// TIA Portal V18 program export: 1 tag tables, 9 data types, 14 data blocks, 112 code blocks (in call order from the OBs), 66 instance data blocks

VAR_GLOBAL   // PLC tag table "Default tag table"
   "mz encoder a" AT %I0.0 : Bool;
   "mz encoder b" AT %I0.1 : Bool;
   "my encoder a" AT %I0.2 : Bool;
   "my encoder b" AT %I0.3 : Bool;
   "mx encoder a" AT %I0.4 : Bool;
   "mx encoder b" AT %I0.5 : Bool;
   "mz up indNOK" AT %I0.6 : Bool;
   "mz down indNOK" AT %I0.7 : Bool;
   "my fwd indNOK" AT %I1.0 : Bool;
   "my rev indNOK" AT %I1.1 : Bool;
   "mx right indNOK" AT %I1.2 : Bool;
   "mx left indNOK" AT %I1.3 : Bool;
   "mo1 tilt fwd indNOK" AT %I1.4 : Bool;
   "mo1 tilt rev indNOK" AT %I1.5 : Bool;
   "na(3)" AT %I1.6 : Bool;
   "na(4)" AT %I1.7 : Bool;
   ai_reserve AT %IW100 : Int;
   "ai_reserve(1)" AT %IW102 : Int;
   hscрезерв AT %ID812 : DInt;
   "hscрезерв(1)" AT %ID816 : DInt;
   "hscрезерв(2)" AT %ID820 : DInt;
   "mz hsc" AT %ID800 : DInt;
   "my hsc" AT %ID804 : DInt;
   "mx hsc" AT %ID808 : DInt;
   "a1_com_di50.0" AT %I50.0 : Bool;
   "a1_com_di50.1" AT %I50.1 : Bool;
   "a1_com_di50.2" AT %I50.2 : Bool;
   "a1_com_di50.3" AT %I50.3 : Bool;
   "a1_com_di50.4" AT %I50.4 : Bool;
   "a1_com_di50.5" AT %I50.5 : Bool;
   "a1_com_di50.6" AT %I50.6 : Bool;
   "a1_com_di50.7" AT %I50.7 : Bool;
   a1_com_di_byte AT %IB50 : Byte;
   "mo1 enc a" AT %I2.0 : Bool;
   "mo1 enc b" AT %I2.1 : Bool;
   "mo2 enc a" AT %I2.2 : Bool;
   "mo2 enc b" AT %I2.3 : Bool;
   "door enc a" AT %I2.4 : Bool;
   "door enc b" AT %I2.5 : Bool;
   "door closed 1 ind NOT" AT %I2.6 : Bool;
   "door open NOK 1 ind" AT %I2.7 : Bool;
   "res i" AT %I3.0 : Bool;
   "mo2 rot home ind" AT %I3.1 : Bool;
   "res i(1)" AT %I3.2 : Bool;
   "air pres ok" AT %I3.3 : Bool;
   "door closed 1 mech Excluded For Xray" AT %I3.4 : Bool;
   "door open 1 mech" AT %I3.5 : Bool;
   "na(1)" AT %I3.6 : Bool;
   "na(2)" AT %I3.7 : Bool;
   "ai_reserve(2)" AT %IW110 : Int;
   "ai_reserve(3)" AT %IW112 : Int;
   "hscрезерв(3)" AT %ID862 : DInt;
   "hscрезерв(4)" AT %ID866 : DInt;
   "hscрезерв(5)" AT %ID870 : DInt;
   "mo1 hsc" AT %ID850 : DInt;
   "mo2 hsc" AT %ID854 : DInt;
   "door hsc" AT %ID858 : DInt;
   "mz up mech" AT %I4.0 : Bool;
   "mz down mech" AT %I4.1 : Bool;
   "CAB phase check OK" AT %I4.2 : Bool;
   lightBarrierOK AT %I4.3 : Bool;
   "my fwd mech" AT %I4.4 : Bool;
   "my rev mech" AT %I4.5 : Bool;
   "xray coler ok" AT %I4.6 : Bool;
   ESTOP_AND_KEY_OK AT %I4.7 : Bool;
   "mx right mech" AT %I5.0 : Bool;
   "mx left mech" AT %I5.1 : Bool;
   "door closed 2 mech Excluded For Xray" AT %I5.2 : Bool;
   "door open 2 mech" AT %I5.3 : Bool;
   "mo1 tilt fwd mech" AT %I5.4 : Bool;
   "mo1 tilt rev mech" AT %I5.5 : Bool;
   "door closed 2 ind NOT" AT %I5.6 : Bool;
   "door open 2 ind NOT" AT %I5.7 : Bool;
   "desk door b close" AT %I6.0 : Bool;
   "desk door b open" AT %I6.1 : Bool;
   "desk o1 tilt b cw" AT %I6.2 : Bool;
   "desk o1 tilt b ccw" AT %I6.3 : Bool;
   "desk b home" AT %I6.4 : Bool;
   "desk b load unload" AT %I6.5 : Bool;
   "desk b laser centr" AT %I6.6 : Bool;
   "res i(3)" AT %I7.0 : Bool;
   "res i(4)" AT %I7.1 : Bool;
   ESTOP_OK AT %I7.2 : Bool;
   Y2_home_esw AT %I7.3 : Bool;
   "shutter open ind" AT %I7.5 : Bool;
   "shutter closed ind" AT %I7.4 : Bool;
   "ESTOP xray OK" AT %I7.6 : Bool;
   "res i(8)" AT %I7.7 : Bool;
   "detector safety ok" AT %I8.0 : Bool;
   "desk o2 rot b fwd" AT %I8.1 : Bool;
   "desk o2 rot b reverse" AT %I8.3 : Bool;
   "desk o2 rot b home" AT %I8.2 : Bool;
   "desk y  b rev" AT %I8.4 : Bool;
   "desk y b fwd" AT %I8.5 : Bool;
   "desk b defect next" AT %I8.6 : Bool;
   "desk b defect prev" AT %I8.7 : Bool;
   "desk sw manual" AT %I9.0 : Bool;
   "desk sw auto" AT %I9.1 : Bool;
   "desk b auto start" AT %I9.2 : Bool;
   "desk b defect mark" AT %I9.3 : Bool;
   "desk x b left" AT %I9.4 : Bool;
   "desk x b right" AT %I9.5 : Bool;
   "desk z up" AT %I9.7 : Bool;
   "desk z down" AT %I9.6 : Bool;
   "remote key activated" AT %I6.7 : Bool;
   "mz up" AT %Q0.1 : Bool;
   "mz down" AT %Q0.2 : Bool;
   "mz up STOP" AT %Q0.3 : Bool;
   "mz down STOP" AT %Q0.4 : Bool;
   "my fwd" AT %Q0.6 : Bool;
   "my rev" AT %Q0.5 : Bool;
   "my fwd STOP" AT %Q0.7 : Bool;
   "my rev STOP" AT %Q1.0 : Bool;
   "shutter out1.1" AT %Q1.1 : Bool;
   "na(5)" AT %Q1.2 : Bool;
   "na(6)" AT %Q1.3 : Bool;
   "na(7)" AT %Q1.4 : Bool;
   "na(8)" AT %Q1.5 : Bool;
   "na(9)" AT %Q1.6 : Bool;
   "na(10)" AT %Q1.7 : Bool;
   "mz up down speed" AT %QW100 : Int;
   "my fwd rev speed" AT %QW102 : Int;
   "a1_com_dq50.0" AT %Q50.0 : Bool;
   "a1_com_dq50.1" AT %Q50.1 : Bool;
   "a1_com_dq50.2" AT %Q50.2 : Bool;
   "a1_com_dq50.3" AT %Q50.3 : Bool;
   "a1_com_dq50.4" AT %Q50.4 : Bool;
   "a1_com_dq50.5" AT %Q50.5 : Bool;
   "a1_com_dq50.6" AT %Q50.6 : Bool;
   "a1_com_dq50.7" AT %Q50.7 : Bool;
   a1_com_dq_byte AT %QB50 : Byte;
   "column yellow" AT %Q2.0 : Bool;
   "column green" AT %Q2.1 : Bool;
   "column red" AT %Q2.2 : Bool;
   "detector power" AT %Q2.3 : Bool;
   "mx right" AT %Q2.5 : Bool;
   "mx left" AT %Q2.6 : Bool;
   "mx right STOP" AT %Q2.7 : Bool;
   "mx left STOP" AT %Q3.0 : Bool;
   "light barrier power" AT %Q3.1 : Bool;
   "res q" AT %Q2.4 : Bool;
   na AT %Q3.2 : Bool;
   na_1 AT %Q3.3 : Bool;
   na_2 AT %Q3.4 : Bool;
   na_3 AT %Q3.5 : Bool;
   na_4 AT %Q3.6 : Bool;
   na_5 AT %Q3.7 : Bool;
   "mx speed right left" AT %QW110 : Int;
   "mo1 tilt speed" AT %QW112 : Int;
   "mo1 tilt fwd" AT %Q4.1 : Bool;
   "mo1 tilt rev" AT %Q4.0 : Bool;
   "mo1 tilt fwd STOP" AT %Q4.2 : Bool;
   "mo1 tilt rev STOP" AT %Q4.3 : Bool;
   "mo2 rot cw" AT %Q4.4 : Bool;
   "mo2 rot ccw" AT %Q4.5 : Bool;
   "mo2 rot cw STOP" AT %Q4.6 : Bool;
   "mo2 rot ccw STOP" AT %Q4.7 : Bool;
   "door close" AT %Q5.0 : Bool;
   "door open" AT %Q5.1 : Bool;
   "door close STOP" AT %Q5.2 : Bool;
   "door open STOP" AT %Q5.3 : Bool;
   "magnet energize" AT %Q5.4 : Bool;
   "laser center energize" AT %Q5.5 : Bool;
   reserve_aq AT %QW118 : Int;
   "reserve_aq(1)" AT %QW120 : Int;
   "mo2 speed" AT %QW114 : Int;
   "door speed" AT %QW116 : Int;
   "desk siren finished" AT %Q6.1 : Bool;
   "desk siren error" AT %Q6.2 : Bool;
   "desk led auto on" AT %Q6.3 : Bool;
   "desk led shutter closed" AT %Q6.4 : Bool;
   "res q(1)" AT %Q6.0 : Bool;
   "remote power supNA" AT %Q6.5 : Bool;
   "res q(2)" AT %Q6.6 : Bool;
   "res q(3)" AT %Q6.7 : Bool;
   "res q(4)" AT %Q7.0 : Bool;
   "res q(5)" AT %Q7.1 : Bool;
   "res q(6)" AT %Q7.2 : Bool;
   "res q(7)" AT %Q7.3 : Bool;
   "res q(8)" AT %Q7.4 : Bool;
   "res q(9)" AT %Q7.5 : Bool;
   "res q(10)" AT %Q7.6 : Bool;
   "res q(11)77" AT %Q7.7 : Bool;
   erCOM_A1 AT %M0.0 : Bool;
   "erCOM_A1(1)" AT %M0.1 : Bool;
   wnDelay AT %M0.2 : Bool;
   MD_CYCLE AT %M0.3 : Bool;
END_VAR
VAR_GLOBAL CONSTANT   // user constants
   "None(1)" : Pip := 65535;
   "Automatic update(1)" : Pip := 0;
   "PIP 1(1)" : Pip := 1;
   "PIP 2(1)" : Pip := 2;
   "PIP 3(1)" : Pip := 3;
   "PIP 4(1)" : Pip := 4;
   "PIP OB Servo(1)" : Pip := 32768;
   "Local~MC(1)" : Hw_SubModule := 51;
   "Local~Exec(1)" : Hw_SubModule := 52;
   "Local(1)" : Hw_SubModule := 49;
   "Local~PROFINET_interface_1(1)" : Hw_Interface := 64;
   "Local~PROFINET_interface_1~Port_1(1)" : Hw_Interface := 65;
   "Local~PROFINET_interface_1~Port_2(1)" : Hw_Interface := 66;
   "Local~HSC_1(1)" : Hw_Hsc := 257;
   "Local~HSC_2(1)" : Hw_Hsc := 258;
   "Local~HSC_3(1)" : Hw_Hsc := 259;
   "Local~HSC_4(1)" : Hw_Hsc := 260;
   "Local~HSC_5(1)" : Hw_Hsc := 261;
   "Local~HSC_6(1)" : Hw_Hsc := 262;
   "Local~AI_2_AQ_2_1(1)" : Hw_SubModule := 263;
   "Local~DI_14_DQ_10_1(1)" : Hw_SubModule := 264;
   "Local~OPC_UA(1)" : Hw_SubModule := 117;
   "Local~Pulse_1(1)" : Hw_Pwm := 265;
   "Local~Pulse_2(1)" : Hw_Pwm := 266;
   "Local~Pulse_3(1)" : Hw_Pwm := 267;
   "Local~Pulse_4(1)" : Hw_Pwm := 268;
   "OB_Main(1)" : OB_PCYCLE := 1;
   "Local~A3_DI_16x24VDC_DQ_16xRelay_1" : Hw_SubModule := 269;
   "Local~A4_AQ_4x14BIT_1" : Hw_SubModule := 270;
   "Local~A5_DI_16x24VDC_DQ_16xRelay_2" : Hw_SubModule := 271;
   "Local~A6_DI_16x24VDC_1" : Hw_SubModule := 272;
   "Local~PROFINET_IO-System(1)" : Hw_IoSystem := 273;
   "A1_slave~PROFINET_interface_1~IODevice(1)" : Hw_Device := 275;
   "A1_slave~PROFINET_interface_1~bool0(1)" : Hw_SubModule := 277;
   "A1_slave~PROFINET_interface_1~bool1(1)" : Hw_SubModule := 278;
   "A1_slave~PROFINET_interface_1~analog0(1)" : Hw_SubModule := 279;
   "A1_slave~PROFINET_interface_1~anolog1(1)" : Hw_SubModule := 280;
   "A1_slave~PROFINET_interface_1~hsc(1)" : Hw_SubModule := 281;
   "A1_slave~PROFINET_interface_1~pulse(1)" : Hw_SubModule := 282;
   "A1_slave~PROFINET_interface_1~comm0(1)" : Hw_SubModule := 283;
   "A1_slave~PROFINET_interface_1~comm1" : Hw_SubModule := 284;
   "Local~Common(1)" : Hw_SubModule := 50;
   "Local~Device(1)" : Hw_Device := 32;
   "Local~Configuration(1)" : Hw_SubModule := 33;
   "OB_Cyclic interrupt" : OB_Cyclic := 30;
END_VAR

TYPE "hmi_home_1"
// stored: IsFailsafeCompliant false
   STRUCT
      pos : Real;
      eF : Bool;
      eR : Bool;
      mF : Bool;
      mR : Bool;
   END_STRUCT;
END_TYPE

TYPE "typeDefectsDB"
// stored: IsFailsafeCompliant false
   STRUCT
      i : Int;
      N : Int;
      N_max : Int := 30;
      pos_AR : Array[1..30] of "typePositions";
   END_STRUCT;
END_TYPE

TYPE "typeGuideAxisBool"
// stored: IsFailsafeCompliant false
   STRUCT
      M1Z : Bool;
      M2Y : Bool;
      M3X : Bool;
      M4O1 : Bool;
      M5O2 : Bool;
      M6doors : Bool;
   END_STRUCT;
END_TYPE

TYPE "typeGuideAxisInt"
// stored: IsFailsafeCompliant false
   STRUCT
      Mot1_RightLeft : Int;
      Mot2_FwdRev : Int;
   END_STRUCT;
END_TYPE

TYPE "typeLimitPack"
// stored: IsFailsafeCompliant false
   STRUCT
      x_min : Real;
      x_max : Real;
      y_min : Real;
      y_max : Real;
   END_STRUCT;
END_TYPE

TYPE "typeMotPara"
// stored: IsFailsafeCompliant false
   STRUCT
      t_acc_50Hz_USER : Real;
      v_absoluteMax_LOGIC : Real;
      dist_absMax_LOGIC : Real;
      v_crawl_USER : Real;
      dist_crawl_USER : Real;
      dist_stop_USER : Real;
      dist_auto_done_LOGIC : Real;
      pos_calib_USER : Real;
      pos_lim_fwd_USER : Real;
      pos_lim_rev_USER : Real;
      v_blind_USER : Real;
      v_manual_USER : Real;
      v_auto_USER : Real;
      t_er : Time := T#3s;
   END_STRUCT;
END_TYPE

TYPE "typePOSMEMcalib"
// stored: IsFailsafeCompliant false
   STRUCT
      MEM : Real;
      offset : Real;
      calibrated : Bool;
   END_STRUCT;
END_TYPE

TYPE "typePositions"
// stored: IsFailsafeCompliant false
   STRUCT
      M1Z : Real;
      M2Y : Real;
      M3X : Real;
      M4O1 : Real;
      M5O2 : Real;
   END_STRUCT;
END_TYPE

TYPE "typeSpotList"
// stored: IsFailsafeCompliant false
   STRUCT
      N : Int;
      pos_AR : Array[1..30] of "typePositions";
   END_STRUCT;
END_TYPE

DATA_BLOCK "TodosDB"   // DB40
{ S7_Optimized_Access := 'TRUE' }
VERSION : 0.1
// stored: AutoNumber true, DBAccessibleFromOPCUA true, IsOnlyStoredInLoadMemory false, IsRetainMemResEnabled false, IsWriteProtectedInAS false, MemoryReserve 100
   VAR
      todoExists : Bool;
   END_VAR
BEGIN
END_DATA_BLOCK

DATA_BLOCK "deleteddb"   // DB60
{ S7_Optimized_Access := 'TRUE' }
VERSION : 0.1
// stored: AutoNumber true, DBAccessibleFromOPCUA true, IsOnlyStoredInLoadMemory false, IsRetainMemResEnabled false, IsWriteProtectedInAS false, MemoryReserve 100
   VAR
      target : Real;
      pos : Real;
      delta : Real;
      prec_au : Real;
      dist_stop : Real;
      arrived : Bool;
      stop_now : Bool;
      distance : Real;
   END_VAR
BEGIN
END_DATA_BLOCK

DATA_BLOCK "teste"   // DB1
{ S7_Optimized_Access := 'TRUE' }
VERSION : 0.1
// stored: AutoNumber true, DBAccessibleFromOPCUA true, IsOnlyStoredInLoadMemory false, IsRetainMemResEnabled false, IsWriteProtectedInAS false, MemoryReserve 100
   VAR
      test : Bool;
      test2 : Bool;
   END_VAR
BEGIN
END_DATA_BLOCK

DATA_BLOCK "Targets"   // DB23
{ S7_Optimized_Access := 'TRUE' }
VERSION : 0.1
// stored: AutoNumber true, DBAccessibleFromOPCUA true, IsOnlyStoredInLoadMemory false, IsRetainMemResEnabled false, IsWriteProtectedInAS false, MemoryReserve 100
   VAR RETAIN
      "A" : Array[1..10] of "typePositions";
   END_VAR
BEGIN
END_DATA_BLOCK

DATA_BLOCK "_POSITIONS_RETAIN"   // DB61
{ S7_Optimized_Access := 'TRUE' }
VERSION : 0.1
// stored: AutoNumber true, DBAccessibleFromOPCUA true, IsOnlyStoredInLoadMemory false, IsRetainMemResEnabled false, IsWriteProtectedInAS false, MemoryReserve 100
   VAR RETAIN
      A1Z { S7_SetPoint := 'True'} : "typePOSMEMcalib";
      A2Y { S7_SetPoint := 'True'} : "typePOSMEMcalib";
      A3X { S7_SetPoint := 'True'} : "typePOSMEMcalib";
      A4O1 { S7_SetPoint := 'True'} : "typePOSMEMcalib";
      A5O2 { S7_SetPoint := 'True'} : "typePOSMEMcalib";
      A6Doors { S7_SetPoint := 'True'} : "typePOSMEMcalib";
   END_VAR
BEGIN
END_DATA_BLOCK

DATA_BLOCK "PC"   // DB69
{ S7_Optimized_Access := 'FALSE'; DB_Accessible_From_OPC_UA := 'FALSE' }
VERSION : 0.1
// stored: AutoNumber false, DBAccessibleFromOPCUA false, IsOnlyStoredInLoadMemory false, IsWriteProtectedInAS false
   VAR
      Keep_alive_fromPLC : Bool;
      X_ray_ready_fromPLC : Bool;
      Image_ready_fromPC : Bool;
      PLC_RESET_Image_ready_fromPC : Bool;
      POS_M1Z : Real;
      POS_M2Y : Real;
      POS_M3X : Real;
      POS_M4O1Tilt : Real;
      POS_M5O2Rot : Real;
   END_VAR
BEGIN
END_DATA_BLOCK

DATA_BLOCK "PARAMs"   // DB17
{ S7_Optimized_Access := 'TRUE' }
VERSION : 0.1
// stored: AutoNumber true, DBAccessibleFromOPCUA true, IsOnlyStoredInLoadMemory false, IsRetainMemResEnabled false, IsWriteProtectedInAS false, MemoryReserve 100
   VAR
      K_min_v : Real := 0.1;
      K_min_dist : Real := 0.003;
      K_dist_fast : Real := 5.0;
   END_VAR
   VAR RETAIN
      M1Z { S7_SetPoint := 'True'} : "typeMotPara";
      M2Y { S7_SetPoint := 'True'} : "typeMotPara";
      M3X { S7_SetPoint := 'True'} : "typeMotPara";
      M4O1 { S7_SetPoint := 'True'} : "typeMotPara";
      M5O2 { S7_SetPoint := 'True'} : "typeMotPara";
      M6Doors { S7_SetPoint := 'True'} : "typeMotPara";
   END_VAR
BEGIN
   M1Z.t_acc_50Hz_USER := 10.0;
   M1Z.v_absoluteMax_LOGIC := 113.3333;
   M1Z.dist_absMax_LOGIC := 581.6667;
   M1Z.v_crawl_USER := 3.0;
   M1Z.dist_crawl_USER := 3.0;
   M1Z.dist_stop_USER := 1.0;
   M1Z.dist_auto_done_LOGIC := 3.0;
   M1Z.pos_calib_USER := 0.0;
   M1Z.pos_lim_fwd_USER := 100.0;
   M1Z.pos_lim_rev_USER := 0.0;
   M1Z.v_blind_USER := 0.0;
   M1Z.v_manual_USER := 0.0;
   M1Z.v_auto_USER := 0.0;
   M1Z.t_er := T#1S;
   M2Y.t_acc_50Hz_USER := 10.0;
   M2Y.v_absoluteMax_LOGIC := 111.6667;
   M2Y.dist_absMax_LOGIC := 608.3333;
   M2Y.v_crawl_USER := 10.0;
   M2Y.dist_crawl_USER := 5.0;
   M2Y.dist_stop_USER := 1.0;
   M2Y.dist_auto_done_LOGIC := 3.0;
   M2Y.pos_calib_USER := 0.0;
   M2Y.pos_lim_fwd_USER := 847.0;
   M2Y.pos_lim_rev_USER := 0.0;
   M2Y.v_blind_USER := 20.0;
   M2Y.v_manual_USER := 50.0;
   M2Y.v_auto_USER := 60.0;
   M2Y.t_er := T#3S;
   M3X.t_acc_50Hz_USER := 3.0;
   M3X.v_absoluteMax_LOGIC := 118.3696;
   M3X.dist_absMax_LOGIC := 185.0543;
   M3X.v_crawl_USER := 5.0;
   M3X.dist_crawl_USER := 2.0;
   M3X.dist_stop_USER := 1.0;
   M3X.dist_auto_done_LOGIC := 3.0;
   M3X.pos_calib_USER := 0.0;
   M3X.pos_lim_fwd_USER := 680.0;
   M3X.pos_lim_rev_USER := 0.0;
   M3X.v_blind_USER := 10.0;
   M3X.v_manual_USER := 50.0;
   M3X.v_auto_USER := 100.0;
   M3X.t_er := T#3S;
   M4O1.t_acc_50Hz_USER := 1.0;
   M4O1.v_absoluteMax_LOGIC := 31.17822;
   M4O1.dist_absMax_LOGIC := 17.08911;
   M4O1.v_crawl_USER := 3.0;
   M4O1.dist_crawl_USER := 2.0;
   M4O1.dist_stop_USER := 1.0;
   M4O1.dist_auto_done_LOGIC := 3.0;
   M4O1.pos_calib_USER := 0.0;
   M4O1.pos_lim_fwd_USER := 5.0;
   M4O1.pos_lim_rev_USER := 0.0;
   M4O1.v_blind_USER := 3.0;
   M4O1.v_manual_USER := 3.0;
   M4O1.v_auto_USER := 1.0;
   M4O1.t_er := T#3S;
   M5O2.t_acc_50Hz_USER := 10.0;
   M5O2.v_absoluteMax_LOGIC := 67.0;
   M5O2.dist_absMax_LOGIC := 345.0;
   M5O2.v_crawl_USER := 2.0;
   M5O2.dist_crawl_USER := 2.0;
   M5O2.dist_stop_USER := 0.2;
   M5O2.dist_auto_done_LOGIC := 0.6;
   M5O2.pos_calib_USER := 0.0;
   M5O2.pos_lim_fwd_USER := 360.0;
   M5O2.pos_lim_rev_USER := 0.0;
   M5O2.v_blind_USER := 30.0;
   M5O2.v_manual_USER := 30.0;
   M5O2.v_auto_USER := 50.0;
   M5O2.t_er := T#3S;
   M6Doors.t_acc_50Hz_USER := 10.0;
   M6Doors.v_absoluteMax_LOGIC := 83.33334;
   M6Doors.dist_absMax_LOGIC := 446.6667;
   M6Doors.v_crawl_USER := 6.0;
   M6Doors.dist_crawl_USER := 6.0;
   M6Doors.dist_stop_USER := 3.0;
   M6Doors.dist_auto_done_LOGIC := 9.0;
   M6Doors.pos_calib_USER := 0.0;
   M6Doors.pos_lim_fwd_USER := 1.0;
   M6Doors.pos_lim_rev_USER := 0.0;
   M6Doors.v_blind_USER := 5.0;
   M6Doors.v_manual_USER := 5.0;
   M6Doors.v_auto_USER := 5.0;
   M6Doors.t_er := T#3S;
END_DATA_BLOCK

DATA_BLOCK "_MAIN_DB"   // DB53
{ S7_Optimized_Access := 'TRUE' }
VERSION : 0.1
// stored: AutoNumber true, DBAccessibleFromOPCUA true, IsOnlyStoredInLoadMemory false, IsRetainMemResEnabled false, IsWriteProtectedInAS false, MemoryReserve 100
   VAR
      CLOCK_S_P_SCAN { ExternalWritable := 'False'; S7_SetPoint := 'True'} : Real := 0.03;
      AllModulesLive : Bool;
      сервисный_ключ : Bool := FALSE;
      медленно : Bool;
      bDefectsReset : Bool;
      bGoToDefectNow : Bool;
      GoToSpotNow : Bool;
      DefectsAllFound_beepResetMe : Bool;
      cycleDoneResetMe : Bool;
      Mot_Targets { S7_SetPoint := 'True'} : "typePositions";
      Mot_Positions { S7_SetPoint := 'True'} : "typePositions";
      MotCalibaratedAr { ExternalWritable := 'False'; S7_SetPoint := 'True'} : "typeGuideAxisBool";
      MotAllCalibrated { ExternalWritable := 'False'; S7_SetPoint := 'True'} : Bool;
      MotArrived { S7_SetPoint := 'True'} : "typeGuideAxisBool";
      MotAllArrived : Bool;
      desk_xAny : Bool;
      buz_alarm_er_count_change : Bool;
      buz_alarm_doorsClosedOpen : Bool;
   END_VAR
   VAR RETAIN
      главный_пульт_медлен : Bool;
   END_VAR
   VAR
      v_auto : Real := 110.0;
      Static_1 : Real := 50.0;
   END_VAR
BEGIN
END_DATA_BLOCK

DATA_BLOCK "Recipe"   // DB76
{ S7_Optimized_Access := 'TRUE' }
VERSION : 0.1
// stored: AutoNumber true, DBAccessibleFromOPCUA true, IsOnlyStoredInLoadMemory false, IsRetainMemResEnabled false, IsWriteProtectedInAS false, MemoryReserve 100
   VAR RETAIN
      RotationStep : Real := 30.0;
   END_VAR
BEGIN
END_DATA_BLOCK

DATA_BLOCK "_ML3_importantPositionsRETAIN"   // DB67
{ S7_Optimized_Access := 'TRUE' }
VERSION : 0.1
// stored: AutoNumber true, DBAccessibleFromOPCUA true, IsOnlyStoredInLoadMemory false, IsRetainMemResEnabled false, IsWriteProtectedInAS false, MemoryReserve 100
   VAR RETAIN
      Load : "typePositions";
      Home : "typePositions";
      Control1 : "typePositions";
      Control2 : "typePositions";
   END_VAR
BEGIN
END_DATA_BLOCK

DATA_BLOCK "_SPOT_DB"   // DB10
{ S7_Optimized_Access := 'TRUE' }
VERSION : 0.1
// stored: AutoNumber true, DBAccessibleFromOPCUA true, IsOnlyStoredInLoadMemory false, IsRetainMemResEnabled false, IsWriteProtectedInAS false, MemoryReserve 100
   VAR
      Spot_i : Int := 0;
      Spot_N_max : Int := 30;
      SpotListNow { S7_SetPoint := 'True'} : "typeSpotList";
   END_VAR
   VAR RETAIN
      Part_selected : Int := 0;
      Part_N : Int;
      Part_N_max : Int := 30;
      Parts { S7_SetPoint := 'True'} : Array[1..10] of "typeSpotList";
   END_VAR
BEGIN
   SpotListNow.N := 4;
   SpotListNow.pos_AR[1].M1Z := 11.0;
   SpotListNow.pos_AR[2].M1Z := 22.0;
   SpotListNow.pos_AR[3].M1Z := 33.0;
   SpotListNow.pos_AR[4..30].M1Z := 0.0;
   SpotListNow.pos_AR[1].M2Y := 11.0;
   SpotListNow.pos_AR[2].M2Y := 22.0;
   SpotListNow.pos_AR[3].M2Y := 33.0;
   SpotListNow.pos_AR[4..30].M2Y := 0.0;
   SpotListNow.pos_AR[1].M3X := 11.0;
   SpotListNow.pos_AR[2].M3X := 22.0;
   SpotListNow.pos_AR[3].M3X := 33.0;
   SpotListNow.pos_AR[4..30].M3X := 0.0;
   SpotListNow.pos_AR[1].M4O1 := 11.0;
   SpotListNow.pos_AR[2].M4O1 := 22.0;
   SpotListNow.pos_AR[3].M4O1 := 33.0;
   SpotListNow.pos_AR[4..30].M4O1 := 0.0;
   SpotListNow.pos_AR[1].M5O2 := 11.0;
   SpotListNow.pos_AR[2].M5O2 := 22.0;
   SpotListNow.pos_AR[3].M5O2 := 33.0;
   SpotListNow.pos_AR[4..30].M5O2 := 0.0;
   Parts[1..10].N := 0;
   Parts[1].pos_AR[1..30].M1Z := 0.0;
   Parts[2].pos_AR[1..30].M1Z := 0.0;
   Parts[3].pos_AR[1..30].M1Z := 0.0;
   Parts[4].pos_AR[1..30].M1Z := 0.0;
   Parts[5].pos_AR[1..30].M1Z := 0.0;
   Parts[6].pos_AR[1..30].M1Z := 0.0;
   Parts[7].pos_AR[1..30].M1Z := 0.0;
   Parts[8].pos_AR[1..30].M1Z := 0.0;
   Parts[9].pos_AR[1..30].M1Z := 0.0;
   Parts[10].pos_AR[1..30].M1Z := 0.0;
   Parts[1].pos_AR[1..30].M2Y := 0.0;
   Parts[2].pos_AR[1..30].M2Y := 0.0;
   Parts[3].pos_AR[1..30].M2Y := 0.0;
   Parts[4].pos_AR[1..30].M2Y := 0.0;
   Parts[5].pos_AR[1..30].M2Y := 0.0;
   Parts[6].pos_AR[1..30].M2Y := 0.0;
   Parts[7].pos_AR[1..30].M2Y := 0.0;
   Parts[8].pos_AR[1..30].M2Y := 0.0;
   Parts[9].pos_AR[1..30].M2Y := 0.0;
   Parts[10].pos_AR[1..30].M2Y := 0.0;
   Parts[1].pos_AR[1..30].M3X := 0.0;
   Parts[2].pos_AR[1..30].M3X := 0.0;
   Parts[3].pos_AR[1..30].M3X := 0.0;
   Parts[4].pos_AR[1..30].M3X := 0.0;
   Parts[5].pos_AR[1..30].M3X := 0.0;
   Parts[6].pos_AR[1..30].M3X := 0.0;
   Parts[7].pos_AR[1..30].M3X := 0.0;
   Parts[8].pos_AR[1..30].M3X := 0.0;
   Parts[9].pos_AR[1..30].M3X := 0.0;
   Parts[10].pos_AR[1..30].M3X := 0.0;
   Parts[1].pos_AR[1..30].M4O1 := 0.0;
   Parts[2].pos_AR[1..30].M4O1 := 0.0;
   Parts[3].pos_AR[1..30].M4O1 := 0.0;
   Parts[4].pos_AR[1..30].M4O1 := 0.0;
   Parts[5].pos_AR[1..30].M4O1 := 0.0;
   Parts[6].pos_AR[1..30].M4O1 := 0.0;
   Parts[7].pos_AR[1..30].M4O1 := 0.0;
   Parts[8].pos_AR[1..30].M4O1 := 0.0;
   Parts[9].pos_AR[1..30].M4O1 := 0.0;
   Parts[10].pos_AR[1..30].M4O1 := 0.0;
   Parts[1].pos_AR[1..30].M5O2 := 0.0;
   Parts[2].pos_AR[1..30].M5O2 := 0.0;
   Parts[3].pos_AR[1..30].M5O2 := 0.0;
   Parts[4].pos_AR[1..30].M5O2 := 0.0;
   Parts[5].pos_AR[1..30].M5O2 := 0.0;
   Parts[6].pos_AR[1..30].M5O2 := 0.0;
   Parts[7].pos_AR[1..30].M5O2 := 0.0;
   Parts[8].pos_AR[1..30].M5O2 := 0.0;
   Parts[9].pos_AR[1..30].M5O2 := 0.0;
   Parts[10].pos_AR[1..30].M5O2 := 0.0;
END_DATA_BLOCK

DATA_BLOCK "LED_HMI"   // DB46
{ S7_Optimized_Access := 'TRUE' }
VERSION : 0.1
// stored: AutoNumber true, DBAccessibleFromOPCUA true, IsOnlyStoredInLoadMemory false, IsRetainMemResEnabled false, IsWriteProtectedInAS false, MemoryReserve 100
   VAR
      test_all : Bool;
   END_VAR
BEGIN
END_DATA_BLOCK

DATA_BLOCK "TAER"   // DB33
{ S7_Optimized_Access := 'TRUE' }
VERSION : 0.1
// stored: AutoNumber true, DBAccessibleFromOPCUA true, IsOnlyStoredInLoadMemory false, IsRetainMemResEnabled false, IsWriteProtectedInAS false, MemoryReserve 100
BEGIN
END_DATA_BLOCK

DATA_BLOCK "_DEFECT_DB"   // DB44
{ S7_Optimized_Access := 'TRUE' }
VERSION : 0.1
// stored: AutoNumber true, DBAccessibleFromOPCUA true, IsOnlyStoredInLoadMemory false, IsRetainMemResEnabled false, IsWriteProtectedInAS false, MemoryReserve 100
   VAR
      DB : "typeDefectsDB";
   END_VAR
BEGIN
END_DATA_BLOCK

ORGANIZATION_BLOCK "Main"   // OB1, LAD, ProgramCycle
{ S7_Optimized_Access := 'TRUE' }
VERSION : 0.1
// stored: AutoNumber true, IsIECCheckEnabled false, SetENOAutomatically false
   VAR_INPUT
      Initial_Call : Bool;
      Remanence : Bool;
   END_VAR
   VAR_TEMP   // added for the SCL form of the ladder/FBD networks
      _w1 : Bool;
      _w2 : Bool;
      _w3 : Bool;
   END_VAR
BEGIN

REGION Network 1
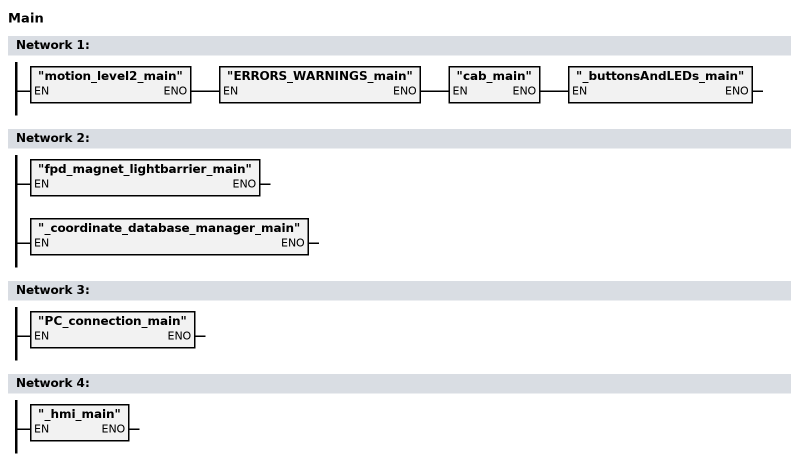
   RUNG wire#powerrail
      "motion_level2_main"()
      "ERRORS_WARNINGS_main"()
      "cab_main"()
      "_buttonsAndLEDs_main"()
   END_RUNG
   // the same network as SCL:
   "motion_level2_main"(ENO => #_w1);
   "ERRORS_WARNINGS_main"(EN := #_w1, ENO => #_w2);
   "cab_main"(EN := #_w2, ENO => #_w3);
   IF #_w3 THEN "_buttonsAndLEDs_main"(); END_IF;
END_REGION

REGION Network 2
   RUNG wire#powerrail
      "fpd_magnet_lightbarrier_main"()
   END_RUNG
   RUNG wire#powerrail
      "_coordinate_database_manager_main"()
   END_RUNG
   // the same network as SCL:
   "fpd_magnet_lightbarrier_main"();
   "_coordinate_database_manager_main"();
END_REGION

REGION Network 3
   RUNG wire#powerrail
      "PC_connection_main"()
   END_RUNG
   // the same network as SCL:
   "PC_connection_main"();
END_REGION

REGION Network 4
   RUNG wire#powerrail
      "_hmi_main"()
   END_RUNG
   // the same network as SCL:
   "_hmi_main"();
END_REGION
END_ORGANIZATION_BLOCK

FUNCTION "motion_level2_main" : Void   // FC22, FBD
{ S7_Optimized_Access := 'TRUE' }
VERSION : 0.1
// stored: AutoNumber true, IsIECCheckEnabled false, SetENOAutomatically false, UDAEnableTagReadback false
   VAR_TEMP
      temp_cycle_run_allowed : Bool;
      man_descrete_button1 : Bool;
      man_descrete_button2 : Bool;
      sel_v_cycle : Bool;
      sel_v_desk : Bool;
      sel_v_rem : Bool;
      place_holder : Bool;
      v_auto : Real;
      v_man : Real;
      go_request : Bool;
      loc_interrupt_semiauto_pbPlaced : Bool;
      queN : UInt;
      Cycle_MotorsGo : Bool;
      авария_расчет_циклических_позиций : Bool;
   END_VAR
BEGIN

REGION Network 2
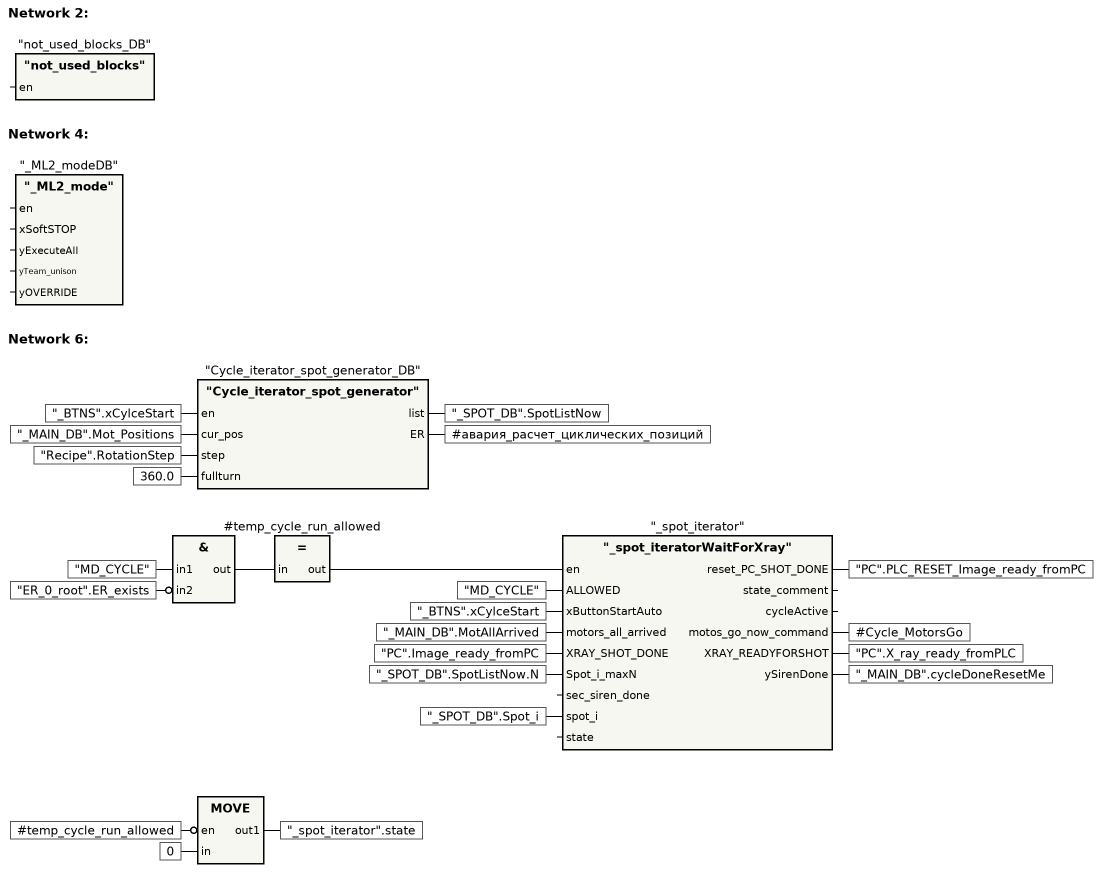
   "not_used_blocks_DB"();   // "not_used_blocks"
END_REGION

REGION Network 4
   "_ML2_modeDB"();   // "_ML2_mode"
END_REGION

REGION Network 6
   IF "_BTNS".xCylceStart THEN
       "Cycle_iterator_spot_generator_DB"(cur_pos := "_MAIN_DB".Mot_Positions,   // "Cycle_iterator_spot_generator"
                               "step" := "Recipe".RotationStep,
                               fullturn := 360.0,
                               list => "_SPOT_DB".SpotListNow,
                               ER => #авария_расчет_циклических_позиций);
   END_IF;
   #temp_cycle_run_allowed := "MD_CYCLE" AND NOT "ER_0_root".ER_exists;
   IF #temp_cycle_run_allowed THEN
       "_spot_iterator"(ALLOWED := "MD_CYCLE",   // "_spot_iteratorWaitForXray"
                        xButtonStartAuto := "_BTNS".xCylceStart,
                        motors_all_arrived := "_MAIN_DB".MotAllArrived,
                        XRAY_SHOT_DONE := "PC".Image_ready_fromPC,
                        Spot_i_maxN := "_SPOT_DB".SpotListNow.N,
                        spot_i := "_SPOT_DB".Spot_i,
                        reset_PC_SHOT_DONE => "PC".PLC_RESET_Image_ready_fromPC,
                        motos_go_now_command => #Cycle_MotorsGo,
                        XRAY_READYFORSHOT => "PC".X_ray_ready_fromPLC,
                        ySirenDone => "_MAIN_DB".cycleDoneResetMe);
   END_IF;
   IF NOT #temp_cycle_run_allowed THEN "_spot_iterator".state := 0; END_IF;
END_REGION

REGION Network 8
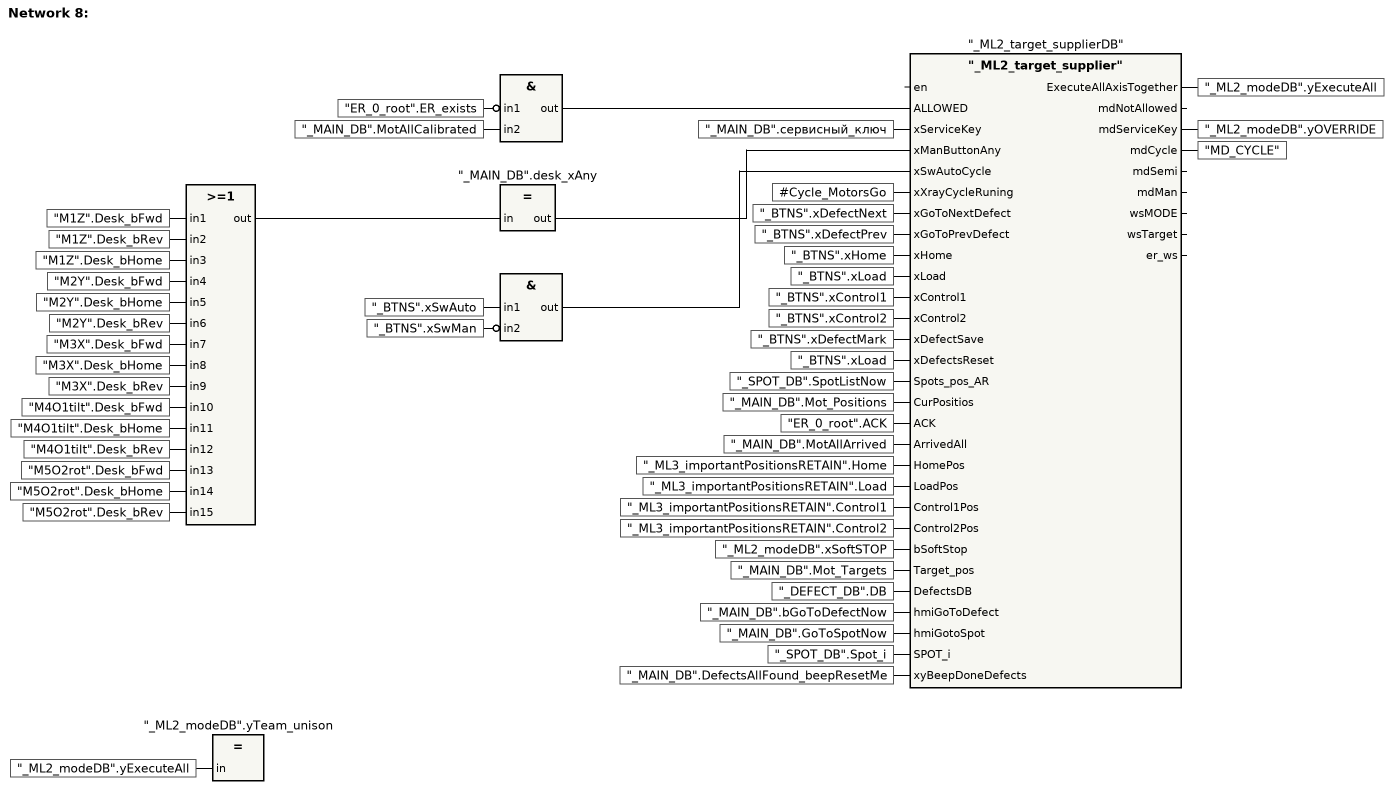
   "_MAIN_DB".desk_xAny := "M1Z".Desk_bFwd OR "M1Z".Desk_bRev OR "M1Z".Desk_bHome OR "M2Y".Desk_bFwd OR "M2Y".Desk_bHome OR "M2Y".Desk_bRev OR "M3X".Desk_bFwd OR "M3X".Desk_bHome OR "M3X".Desk_bRev OR "M4O1tilt".Desk_bFwd OR "M4O1tilt".Desk_bHome OR "M4O1tilt".Desk_bRev OR "M5O2rot".Desk_bFwd OR "M5O2rot".Desk_bHome OR "M5O2rot".Desk_bRev;
   "_ML2_target_supplierDB"(ALLOWED := NOT "ER_0_root".ER_exists AND "_MAIN_DB".MotAllCalibrated,   // "_ML2_target_supplier"
                           xServiceKey := "_MAIN_DB".сервисный_ключ,
                           xManButtonAny := "_MAIN_DB".desk_xAny,
                           xSwAutoCycle := "_BTNS".xSwAuto AND NOT "_BTNS".xSwMan,
                           xXrayCycleRuning := #Cycle_MotorsGo,
                           xGoToNextDefect := "_BTNS".xDefectNext,
                           xGoToPrevDefect := "_BTNS".xDefectPrev,
                           xHome := "_BTNS".xHome,
                           xLoad := "_BTNS".xLoad,
                           xControl1 := "_BTNS".xControl1,
                           xControl2 := "_BTNS".xControl2,
                           xDefectSave := "_BTNS".xDefectMark,
                           xDefectsReset := "_BTNS".xLoad,
                           Spots_pos_AR := "_SPOT_DB".SpotListNow,
                           CurPositios := "_MAIN_DB".Mot_Positions,
                           ACK := "ER_0_root".ACK,
                           ArrivedAll := "_MAIN_DB".MotAllArrived,
                           HomePos := "_ML3_importantPositionsRETAIN".Home,
                           LoadPos := "_ML3_importantPositionsRETAIN".Load,
                           Control1Pos := "_ML3_importantPositionsRETAIN".Control1,
                           Control2Pos := "_ML3_importantPositionsRETAIN".Control2,
                           bSoftStop := "_ML2_modeDB".xSoftSTOP,
                           Target_pos := "_MAIN_DB".Mot_Targets,
                           DefectsDB := "_DEFECT_DB".DB,
                           hmiGoToDefect := "_MAIN_DB".bGoToDefectNow,
                           hmiGotoSpot := "_MAIN_DB".GoToSpotNow,
                           SPOT_i := "_SPOT_DB".Spot_i,
                           xyBeepDoneDefects := "_MAIN_DB".DefectsAllFound_beepResetMe,
                           ExecuteAllAxisTogether => "_ML2_modeDB".yExecuteAll,
                           mdServiceKey => "_ML2_modeDB".yOVERRIDE,
                           mdCycle => "MD_CYCLE");
   "_ML2_modeDB".yTeam_unison := "_ML2_modeDB".yExecuteAll;
END_REGION

REGION Network 11
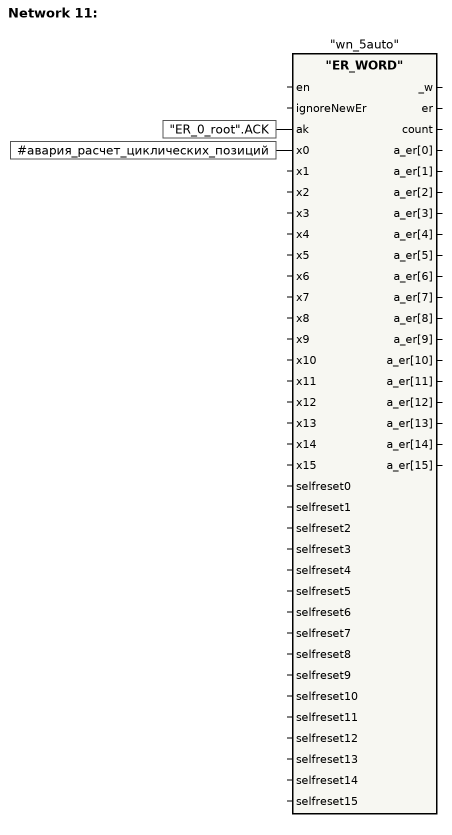
   "wn_5auto"(ak := "ER_0_root".ACK, x0 := #авария_расчет_циклических_позиций);   // "ER_WORD"
END_REGION
END_FUNCTION

FUNCTION_BLOCK "not_used_blocks"   // FB48, FBD
{ S7_Optimized_Access := 'TRUE' }
VERSION : 0.1
// stored: AutoNumber true, IsIECCheckEnabled false, IsRetainMemResEnabled false, MemoryReserve 100, SetENOAutomatically false, UDAEnableTagReadback false
   VAR
      isMultiturn : Bool;
      MultiTurnGoesFwdOnly : Bool;
      SET_SPD_ABS : Real;
      POS : Real;
      TARGET : Real;
      par_lim_fwd : Real;
      par_lim_rev : Real;
      par_spd_absmax : Real;
      par_dist_absMax : Real;
      par_spd_crawl : Real;
      par_dist_crawl : Real;
      par_dist_stop : Real;
      speed_limited_by_target : Real;
      ER : Bool;
      ER_w : WString;
      mot_universal_arrived_missed_Instance { S7_SetPoint := 'True'} : "mot_universal_arrived_missed";
      was_set : Bool;
   END_VAR
   VAR_TEMP
      rtyui1 : Bool;
   END_VAR
BEGIN

REGION Network 2
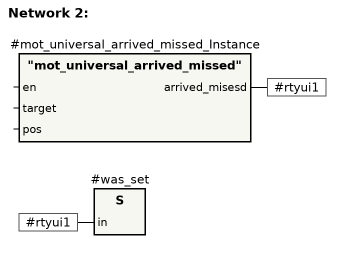
   #mot_universal_arrived_missed_Instance(arrived_misesd => #rtyui1);   // "mot_universal_arrived_missed"
   IF #rtyui1 THEN #was_set := TRUE; END_IF;
END_REGION
END_FUNCTION_BLOCK

FUNCTION_BLOCK "mot_universal_arrived_missed"   // FB70, FBD
{ S7_Optimized_Access := 'TRUE' }
VERSION : 0.1
// stored: AutoNumber true, IsIECCheckEnabled false, IsRetainMemResEnabled false, MemoryReserve 100, SetENOAutomatically false, UDAEnableTagReadback false
   VAR_INPUT
      target : Real;
      pos : Real;
   END_VAR
   VAR_OUTPUT
      arrived_misesd : Bool;
   END_VAR
   VAR
      target_was : Real;
      dir_to_target_pos : Bool;
      dir_to_target_pos_was : Bool;
   END_VAR
BEGIN

REGION Network 2 (SCL)
   #dir_to_target_pos := #pos < #target;

   IF #target = #target_was THEN
       #arrived_misesd := #dir_to_target_pos XOR #dir_to_target_pos_was;
   ELSE
       #arrived_misesd := false;

   END_IF;

   #target_was := #target;
   #dir_to_target_pos_was := #dir_to_target_pos;
END_REGION
END_FUNCTION_BLOCK

FUNCTION_BLOCK "_ML2_mode"   // FB45, FBD
{ S7_Optimized_Access := 'TRUE' }
VERSION : 0.1
// stored: AutoNumber true, IsIECCheckEnabled false, IsRetainMemResEnabled false, MemoryReserve 100, SetENOAutomatically false, UDAEnableTagReadback false
   VAR_IN_OUT
      xSoftSTOP : Bool;
      yExecuteAll : Bool;
      yTeam_unison : Bool;
      yOVERRIDE : Bool;
   END_VAR
BEGIN
END_FUNCTION_BLOCK

FUNCTION_BLOCK "Cycle_iterator_spot_generator"   // FB78, FBD
{ S7_Optimized_Access := 'TRUE' }
VERSION : 0.1
// stored: AutoNumber true, IsIECCheckEnabled false, IsRetainMemResEnabled false, MemoryReserve 100, SetENOAutomatically false, UDAEnableTagReadback false
   VAR_INPUT
      cur_pos : "typePositions";
      "step" : Real;
      fullturn : Real;
   END_VAR
   VAR_OUTPUT
      list : "typeSpotList";
      ER : Bool;
   END_VAR
   VAR
      j : Int;
   END_VAR
   VAR_TEMP
      N : Real;
   END_VAR
BEGIN

REGION Network 1 (SCL)
   #N := #fullturn / #step;

   #list.N := DINT_TO_INT(CEIL(#N));
END_REGION

REGION Network 2 (SCL)

   #ER := FALSE;

   IF #fullturn > 0.0 AND #step > 0 AND #step < #fullturn AND #list.N > 1 AND #list.N <= "_SPOT_DB".Spot_N_max THEN
       FOR #j := 1 TO #list.N DO
           #list.pos_AR[#j] := #cur_pos;
           #list.pos_AR[#j].M5O2 := #step * INT_TO_REAL(#j - 1);
       END_FOR;

   ELSE
       #ER := true;
   END_IF;
END_REGION
END_FUNCTION_BLOCK

FUNCTION_BLOCK "_spot_iteratorWaitForXray"   // FB33, FBD
{ S7_Optimized_Access := 'TRUE' }
VERSION : 0.1
// stored: AutoNumber true, IsIECCheckEnabled false, IsRetainMemResEnabled false, MemoryReserve 100, SetENOAutomatically false, UDAEnableTagReadback false
   VAR_INPUT
      ALLOWED : Bool;
      xButtonStartAuto : Bool;
      motors_all_arrived : Bool;
      XRAY_SHOT_DONE : Bool;
      Spot_i_maxN : Int;
      sec_siren_done : Real := 2.0;
   END_VAR
   VAR_OUTPUT
      reset_PC_SHOT_DONE : Bool;
      state_comment : WString;
      cycleActive : Bool;
      motos_go_now_command : Bool;
      XRAY_READYFORSHOT : Bool;
      ySirenDone : Bool;
   END_VAR
   VAR_IN_OUT
      spot_i : Int;
      state : UInt;
   END_VAR
   VAR
      pt_siren_done { ExternalAccessible := 'False'; ExternalVisible := 'False'; ExternalWritable := 'False'} : Time := T#1s;
      mem1 : Bool;
      mem2 : Bool;
      tons12 { S7_SetPoint := 'True'} : TON_TIME;
      tons20 { S7_SetPoint := 'True'} : TON_TIME;
      tons10 { S7_SetPoint := 'True'} : TON_TIME;
      pt_xray_stuck_in_done { ExternalAccessible := 'False'; ExternalVisible := 'False'; ExternalWritable := 'False'} : Time := T#1s;
      pt_mot_delay : Time := T#100ms;
      tons20a { S7_SetPoint := 'True'} : TON_TIME;
      tons24 { S7_SetPoint := 'True'} : TON_TIME;
      mem3 : Bool;
   END_VAR
   VAR_TEMP
      temp_be_going_to_next_SPOT : Bool;
      temp_be_going_home : Bool;
      reset_pc_shot_done_s20 : Bool;
      reset_pc_shot_done_s23 : Bool;
      queEndReached : Bool;
   END_VAR
   VAR CONSTANT
      s0wait : UInt := 0;
      s20NextPositionGoCommand : UInt := 20;
      s21NextPositionGoing : UInt := 21;
      s22NextPositionArrivedWaitingForXrayPicture : UInt := 22;
      s23NextPositionIncrement : UInt := 23;
      s24NextPositionDone : UInt := 24;
      wstrings00wait : WString := WSTRING#'Ожидание';
      wstrings20NextPositionGoCommand_1 : WString := WSTRING#'Движение к следующей позиции';
      wstrings21NextPositionGoing_1 : WString := WSTRING#'Движение к следующей позиции';
      wstrings22NextPositionArrivedWaitingForXrayPicture_1 : WString := WSTRING#'ожидание снимка';
      wstrings23NextPositionIncrement_1 : WString := WSTRING#'увеличение индекса позиции';
      wstrings24NextPositionDone_1 : WString := WSTRING#'Цикл завершен';
      CELL_INDEX_HOME : UInt := 1;
      Spot_index_start : UInt := 1;
   END_VAR
   VAR_TEMP   // added for the SCL form of the ladder/FBD networks
      _w1 : Bool;
      _w2 : Bool;
      _w3 : Bool;
      _w4 : Bool;
   END_VAR
BEGIN

REGION Network 3
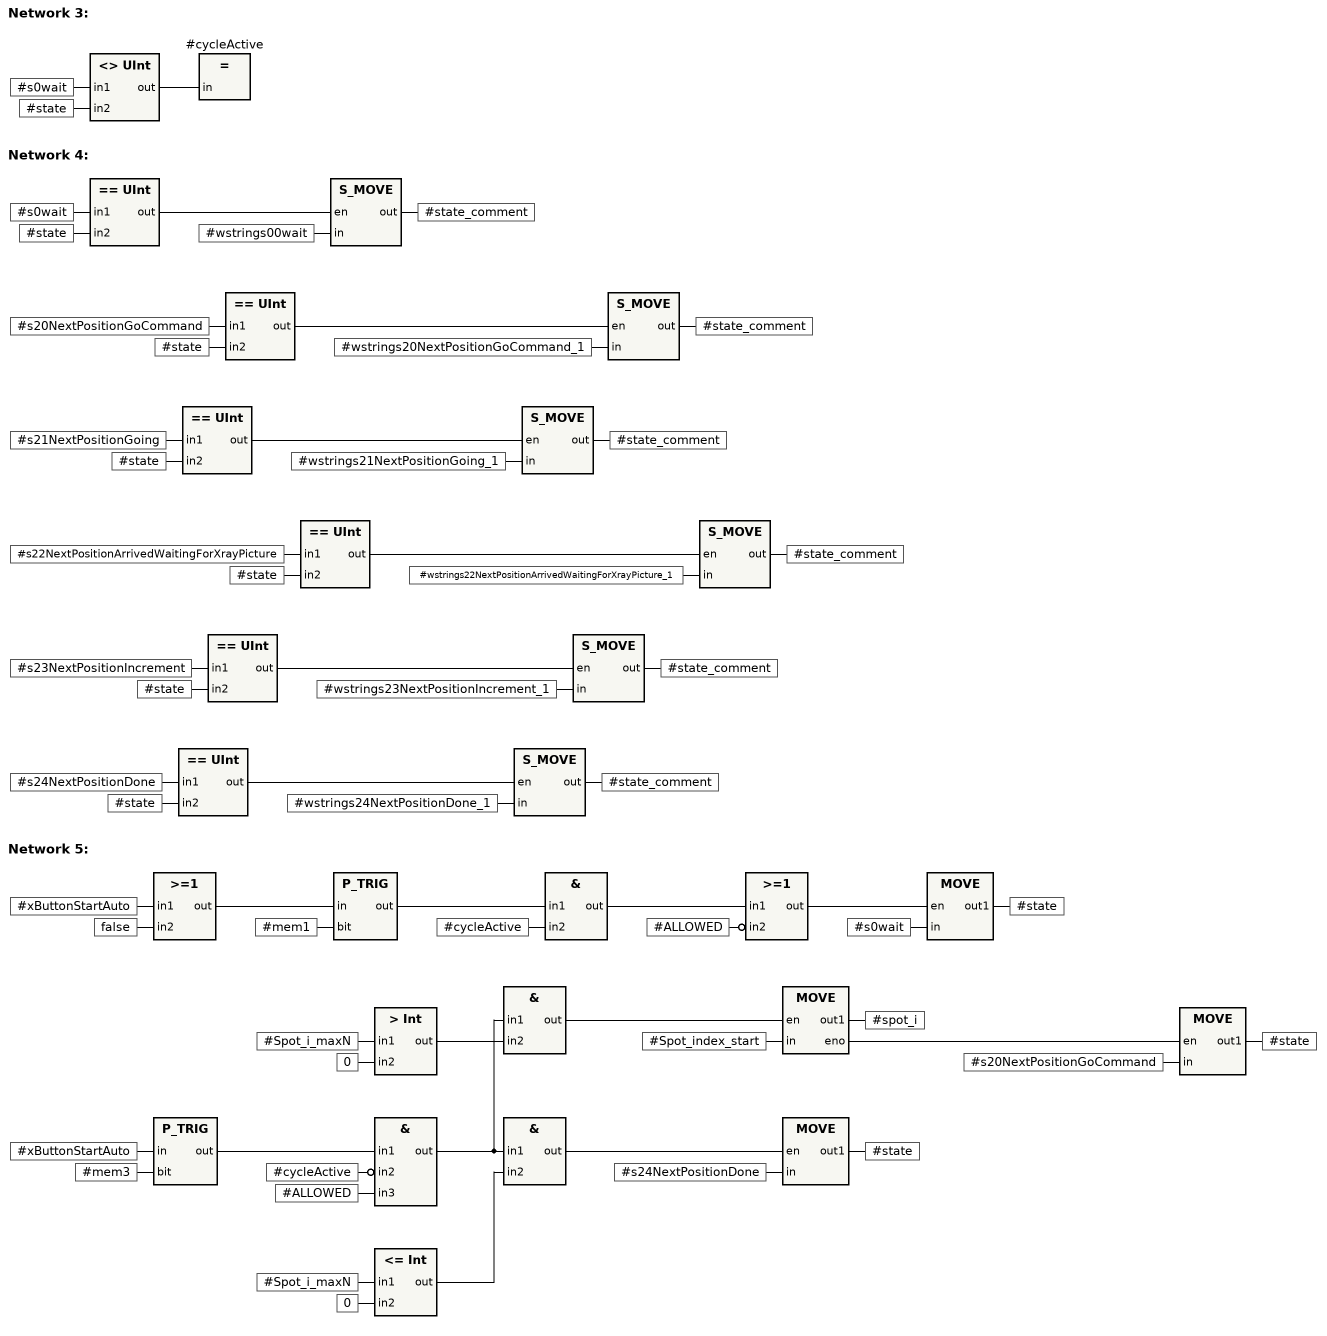
   #cycleActive := #s0wait <> #state;
END_REGION

REGION Network 4
   IF #s0wait = #state THEN #state_comment := #wstrings00wait; END_IF;
   IF #s20NextPositionGoCommand = #state THEN #state_comment := #wstrings20NextPositionGoCommand_1; END_IF;
   IF #s21NextPositionGoing = #state THEN #state_comment := #wstrings21NextPositionGoing_1; END_IF;
   IF #s22NextPositionArrivedWaitingForXrayPicture = #state THEN
       #state_comment := #wstrings22NextPositionArrivedWaitingForXrayPicture_1;
   END_IF;
   IF #s23NextPositionIncrement = #state THEN #state_comment := #wstrings23NextPositionIncrement_1; END_IF;
   IF #s24NextPositionDone = #state THEN #state_comment := #wstrings24NextPositionDone_1; END_IF;
END_REGION

REGION Network 5
   #_w1 := #xButtonStartAuto OR false;
   #_w2 := #_w1 AND NOT #mem1;   // rising edge
   #mem1 := #_w1;
   IF (#_w2 AND #cycleActive) OR NOT #ALLOWED THEN #state := #s0wait; END_IF;
   #_w3 := #xButtonStartAuto AND NOT #mem3;   // rising edge
   #mem3 := #xButtonStartAuto;
   #_w4 := #_w3 AND NOT #cycleActive AND #ALLOWED;
   IF #_w4 AND (#Spot_i_maxN > 0) THEN
       #spot_i := #Spot_index_start;
       #state := #s20NextPositionGoCommand;
   END_IF;
   IF #_w4 AND (#Spot_i_maxN <= 0) THEN #state := #s24NextPositionDone; END_IF;
END_REGION

REGION Network 6
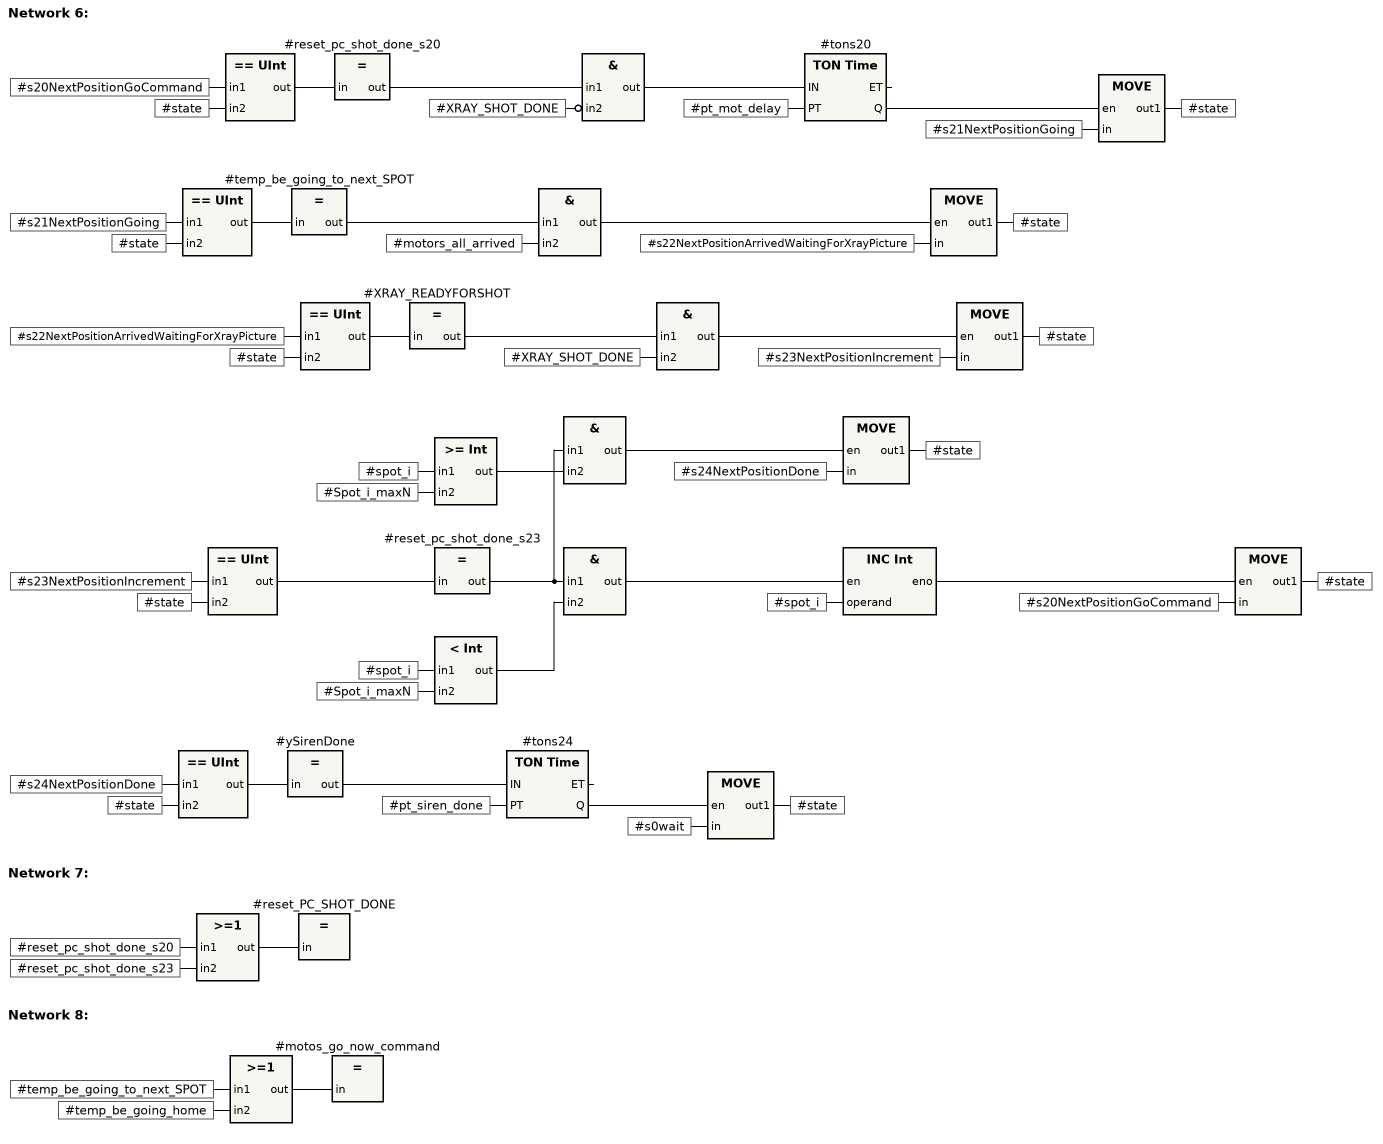
   #reset_pc_shot_done_s20 := #s20NextPositionGoCommand = #state;
   #tons20(IN := #reset_pc_shot_done_s20 AND NOT #XRAY_SHOT_DONE, PT := #pt_mot_delay);   // TON
   IF #tons20.Q THEN #state := #s21NextPositionGoing; END_IF;
   #temp_be_going_to_next_SPOT := #s21NextPositionGoing = #state;
   IF #temp_be_going_to_next_SPOT AND #motors_all_arrived THEN
       #state := #s22NextPositionArrivedWaitingForXrayPicture;
   END_IF;
   #XRAY_READYFORSHOT := #s22NextPositionArrivedWaitingForXrayPicture = #state;
   IF #XRAY_READYFORSHOT AND #XRAY_SHOT_DONE THEN #state := #s23NextPositionIncrement; END_IF;
   #reset_pc_shot_done_s23 := #s23NextPositionIncrement = #state;
   IF #reset_pc_shot_done_s23 AND (#spot_i >= #Spot_i_maxN) THEN #state := #s24NextPositionDone; END_IF;
   #_w1 := #reset_pc_shot_done_s23 AND (#spot_i < #Spot_i_maxN);
   IF #_w1 THEN
       #spot_i := #spot_i + 1;
       #state := #s20NextPositionGoCommand;
   END_IF;
   #ySirenDone := #s24NextPositionDone = #state;
   #tons24(IN := #ySirenDone, PT := #pt_siren_done);   // TON
   IF #tons24.Q THEN #state := #s0wait; END_IF;
END_REGION

REGION Network 7
   #reset_PC_SHOT_DONE := #reset_pc_shot_done_s20 OR #reset_pc_shot_done_s23;
END_REGION

REGION Network 8
   #motos_go_now_command := #temp_be_going_to_next_SPOT OR #temp_be_going_home;
END_REGION

REGION Network 9 (SCL)
   #pt_siren_done := REAL_TO_DINT(#sec_siren_done * 1000);
END_REGION
END_FUNCTION_BLOCK

FUNCTION_BLOCK "_ML2_target_supplier"   // FB29, FBD
{ S7_Optimized_Access := 'TRUE' }
VERSION : 0.1
// stored: AutoNumber true, IsIECCheckEnabled false, IsRetainMemResEnabled false, MemoryReserve 100, SetENOAutomatically false, UDAEnableTagReadback false
   VAR_INPUT
      ALLOWED : Bool;
      xServiceKey : Bool;
      xManButtonAny : Bool;
      xSwAutoCycle : Bool;
      xXrayCycleRuning : Bool;
      xGoToNextDefect : Bool;
      xGoToPrevDefect : Bool;
      xHome : Bool;
      xLoad : Bool;
      xControl1 : Bool;
      xControl2 : Bool;
      xDefectSave : Bool;
      xDefectsReset : Bool;
      Spots_pos_AR : "typeSpotList";
      CurPositios : "typePositions";
      ACK : Bool;
      ArrivedAll : Bool;
      HomePos : "typePositions";
      LoadPos : "typePositions";
      Control1Pos : "typePositions";
      Control2Pos : "typePositions";
      bSoftStop : Bool;
   END_VAR
   VAR_OUTPUT
      ExecuteAllAxisTogether : Bool;
      mdNotAllowed : Bool;
      mdServiceKey : Bool;
      mdCycle : Bool;
      mdSemi : Bool;
      mdMan : Bool;
      wsMODE : WString;
      wsTarget : WString;
      er_ws : WString;
   END_VAR
   VAR_IN_OUT
      Target_pos : "typePositions";
      DefectsDB : "typeDefectsDB";
      hmiGoToDefect : Bool;
      hmiGotoSpot : Bool;
      SPOT_i : Int;
      xyBeepDoneDefects : Bool;
   END_VAR
   VAR
      def_util_db { S7_SetPoint := 'True'} : "defects_util";
      mdSemi_was : Bool;
      st_goToDefectNow : Bool;
      q0_auto : Bool;
      q00_semi : Bool;
      q1_spot : Bool;
      p1_spot : Bool;
      q2_defect : Bool;
      p2_defect : Bool;
      q99_none : Bool;
      q_auto_waiting : Bool;
      block1 { S7_SetPoint := 'True'} : "_ML2_ts_block1";
      p3_home : Bool;
      q3_home : Bool;
      p4_load : Bool;
      q4_load : Bool;
      p5_control1 : Bool;
      q5_control1 : Bool;
      p6_control2 : Bool;
      q6_control2 : Bool;
   END_VAR
   VAR_TEMP
      locSpot_i_winBounds : Bool;
      locDefect_i_winBounds : Bool;
   END_VAR
   VAR CONSTANT
      wm_not_allowed : WString := WSTRING#'Авария';
      wm_cycle : WString := WSTRING#'Автомат';
      wm_service_key : WString := WSTRING#'Сервисный Режим';
      wm_semi_auto : WString := WSTRING#'Полуавтомат';
      wm_man : WString := WSTRING#'Ручной';
      wt00_off : WString := WSTRING#'цель не задана';
      wt0_cycle : WString := WSTRING#'автомат к точке';
      wt1_spot_man : WString := WSTRING#'ручной к точке';
      wt2_defect : WString := WSTRING#'к дефекту';
      wt3_Home : WString := WSTRING#'к домашней позиции';
      wt4_load : WString := WSTRING#'к позиции загрузки';
      wt5_Control1 : WString := WSTRING#'к первому шву';
      wt6_Control2 : WString := WSTRING#'ко второму шву';
      erws_spot_i_lt0_gt_n : WString := WSTRING#'erws_spot_i_lt0_gt_n';
      erws_defect_i_lt0_gt_n_1 : WString := WSTRING#'erws_defecti_lt0_gt_n';
   END_VAR
   VAR_TEMP   // added for the SCL form of the ladder/FBD networks
      _w1 : Bool;
   END_VAR
BEGIN

REGION Network 1
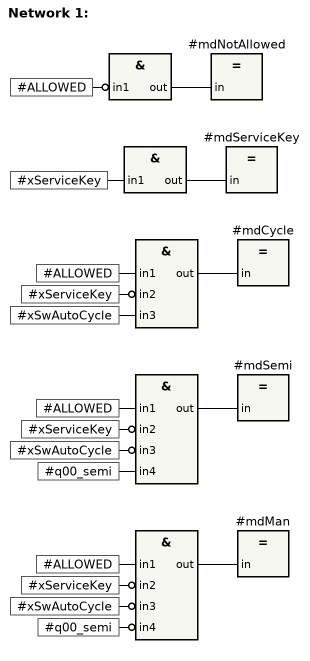
   #mdNotAllowed := NOT #ALLOWED;
   #mdServiceKey := #xServiceKey;
   #mdCycle := #ALLOWED AND NOT #xServiceKey AND #xSwAutoCycle;
   #mdSemi := #ALLOWED AND NOT #xServiceKey AND NOT #xSwAutoCycle AND #q00_semi;
   #mdMan := #ALLOWED AND NOT #xServiceKey AND NOT #xSwAutoCycle AND NOT #q00_semi;
END_REGION

REGION Network 2
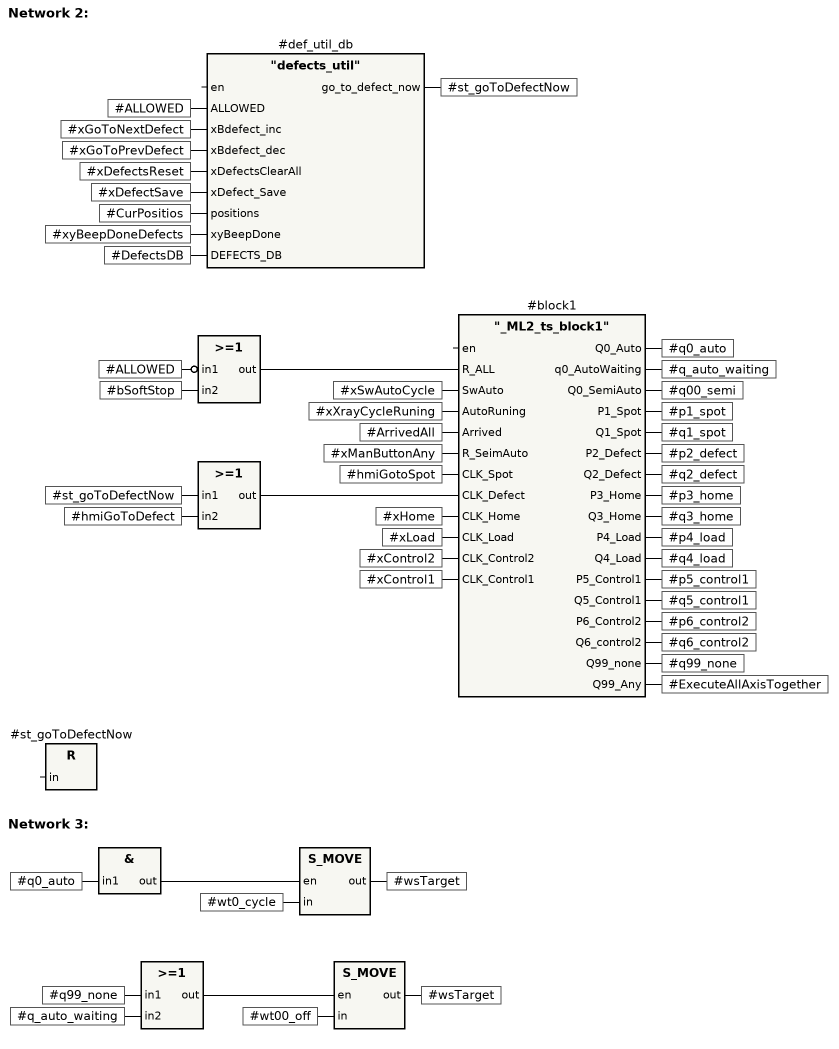
   #def_util_db(ALLOWED := #ALLOWED,   // "defects_util"
                xBdefect_inc := #xGoToNextDefect,
                xBdefect_dec := #xGoToPrevDefect,
                xDefectsClearAll := #xDefectsReset,
                xDefect_Save := #xDefectSave,
                positions := #CurPositios,
                xyBeepDone := #xyBeepDoneDefects,
                DEFECTS_DB := #DefectsDB,
                go_to_defect_now => #st_goToDefectNow);
   #block1(R_ALL := NOT #ALLOWED OR #bSoftStop,   // "_ML2_ts_block1"
           SwAuto := #xSwAutoCycle,
           AutoRuning := #xXrayCycleRuning,
           Arrived := #ArrivedAll,
           R_SeimAuto := #xManButtonAny,
           CLK_Spot := #hmiGotoSpot,
           CLK_Defect := #st_goToDefectNow OR #hmiGoToDefect,
           CLK_Home := #xHome,
           CLK_Load := #xLoad,
           CLK_Control2 := #xControl2,
           CLK_Control1 := #xControl1,
           Q0_Auto => #q0_auto,
           q0_AutoWaiting => #q_auto_waiting,
           Q0_SemiAuto => #q00_semi,
           P1_Spot => #p1_spot,
           Q1_Spot => #q1_spot,
           P2_Defect => #p2_defect,
           Q2_Defect => #q2_defect,
           P3_Home => #p3_home,
           Q3_Home => #q3_home,
           P4_Load => #p4_load,
           Q4_Load => #q4_load,
           P5_Control1 => #p5_control1,
           Q5_Control1 => #q5_control1,
           P6_Control2 => #p6_control2,
           Q6_control2 => #q6_control2,
           Q99_none => #q99_none,
           Q99_Any => #ExecuteAllAxisTogether);
   #st_goToDefectNow := FALSE;
END_REGION

REGION Network 3
   IF #q0_auto THEN #wsTarget := #wt0_cycle; END_IF;
   IF #q99_none OR #q_auto_waiting THEN #wsTarget := #wt00_off; END_IF;
END_REGION

REGION Network 4
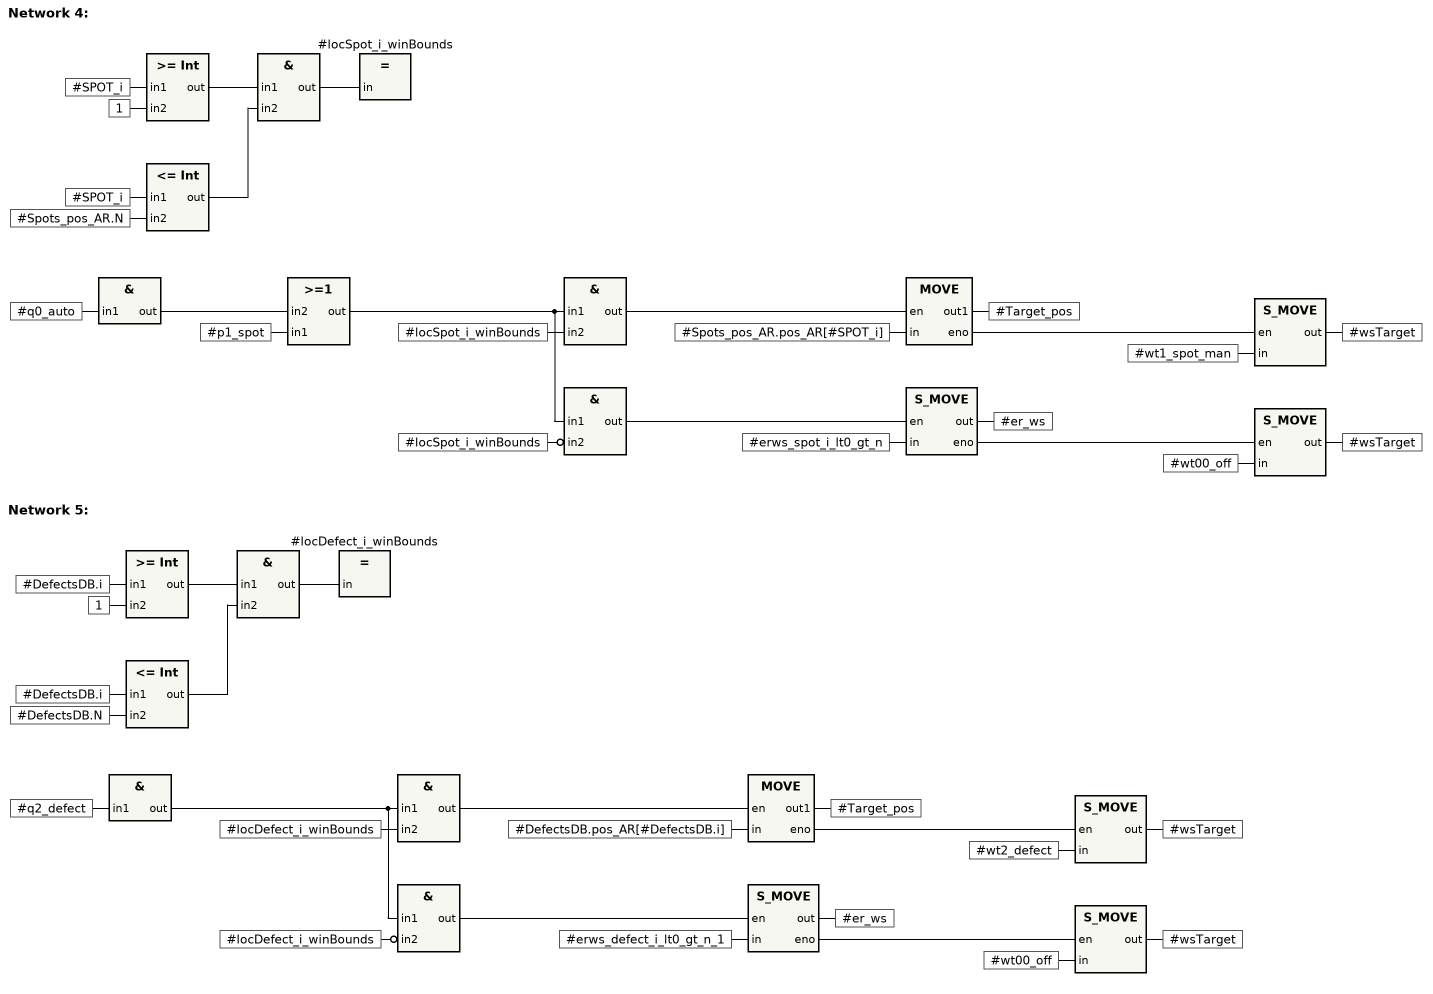
   #locSpot_i_winBounds := (#SPOT_i >= 1) AND (#SPOT_i <= #Spots_pos_AR.N);
   #_w1 := #q0_auto OR #p1_spot;
   IF #_w1 AND #locSpot_i_winBounds THEN
       #Target_pos := #Spots_pos_AR.pos_AR[#SPOT_i];
       #wsTarget := #wt1_spot_man;
   END_IF;
   IF #_w1 AND NOT #locSpot_i_winBounds THEN
       #er_ws := #erws_spot_i_lt0_gt_n;
       #wsTarget := #wt00_off;
   END_IF;
END_REGION

REGION Network 5
   #locDefect_i_winBounds := (#DefectsDB.i >= 1) AND (#DefectsDB.i <= #DefectsDB.N);
   IF #q2_defect AND #locDefect_i_winBounds THEN
       #Target_pos := #DefectsDB.pos_AR[#DefectsDB.i];
       #wsTarget := #wt2_defect;
   END_IF;
   IF #q2_defect AND NOT #locDefect_i_winBounds THEN
       #er_ws := #erws_defect_i_lt0_gt_n_1;
       #wsTarget := #wt00_off;
   END_IF;
END_REGION

REGION Network 6
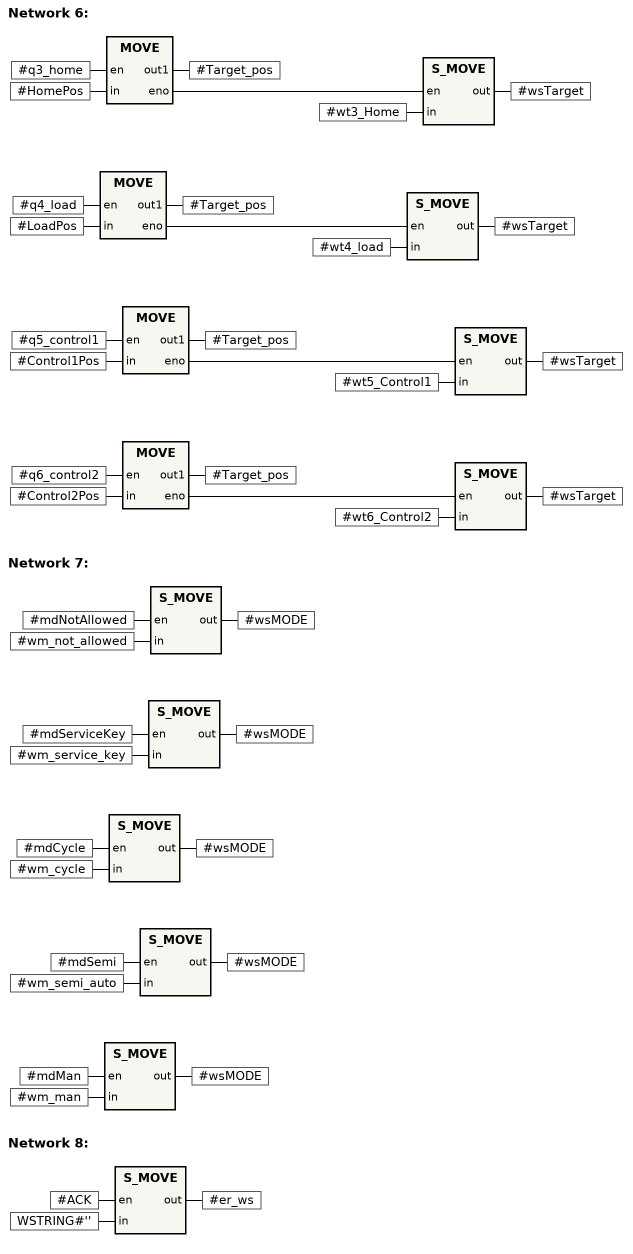
   IF #q3_home THEN
       #Target_pos := #HomePos;
       #wsTarget := #wt3_Home;
   END_IF;
   IF #q4_load THEN
       #Target_pos := #LoadPos;
       #wsTarget := #wt4_load;
   END_IF;
   IF #q5_control1 THEN
       #Target_pos := #Control1Pos;
       #wsTarget := #wt5_Control1;
   END_IF;
   IF #q6_control2 THEN
       #Target_pos := #Control2Pos;
       #wsTarget := #wt6_Control2;
   END_IF;
END_REGION

REGION Network 7
   IF #mdNotAllowed THEN #wsMODE := #wm_not_allowed; END_IF;
   IF #mdServiceKey THEN #wsMODE := #wm_service_key; END_IF;
   IF #mdCycle THEN #wsMODE := #wm_cycle; END_IF;
   IF #mdSemi THEN #wsMODE := #wm_semi_auto; END_IF;
   IF #mdMan THEN #wsMODE := #wm_man; END_IF;
END_REGION

REGION Network 8
   IF #ACK THEN #er_ws := WSTRING#''; END_IF;
END_REGION
END_FUNCTION_BLOCK

FUNCTION_BLOCK "defects_util"   // FB31, FBD
{ S7_Optimized_Access := 'TRUE' }
VERSION : 0.1
// stored: AutoNumber true, IsIECCheckEnabled false, IsRetainMemResEnabled false, MemoryReserve 100, SetENOAutomatically false, UDAEnableTagReadback false
   VAR_INPUT
      ALLOWED : Bool;
      xBdefect_inc : Bool;
      xBdefect_dec : Bool;
      xDefectsClearAll : Bool;
      xDefect_Save : Bool;
      positions : "typePositions";
   END_VAR
   VAR_OUTPUT
      go_to_defect_now : Bool;
   END_VAR
   VAR_IN_OUT
      xyBeepDone : Bool;
      DEFECTS_DB : "typeDefectsDB";
   END_VAR
   VAR
      mem1 : Bool;
      mem2 : Bool;
      xdefect_dec_was : Bool;
      xdefect_inc_was : Bool;
      xDefect_Save_was : Bool;
      xDefectsClearAll_was : Bool;
   END_VAR
BEGIN

REGION Network 1 (SCL)
   IF #ALLOWED THEN
       IF #xBdefect_inc AND NOT #xdefect_inc_was THEN
           IF #DEFECTS_DB.N >0 THEN
               IF #DEFECTS_DB.i < #DEFECTS_DB.N THEN
                   #DEFECTS_DB.i := #DEFECTS_DB.i + 1;
                   #go_to_defect_now := true;
               ELSE
                   #xyBeepDone := true;
                   #DEFECTS_DB.i := #DEFECTS_DB.N;
               END_IF;
               #xyBeepDone := true;
           END_IF;
       END_IF;


       IF #xBdefect_dec AND NOT #xdefect_dec_was THEN
           IF #DEFECTS_DB.i > 1 THEN
               #DEFECTS_DB.i := #DEFECTS_DB.i - 1;
               #go_to_defect_now := true;
           ELSE
               #DEFECTS_DB.i :=  1;
               #xyBeepDone := true;
           END_IF;
       END_IF;
       IF NOT #xBdefect_inc AND NOT #xBdefect_dec THEN
           #go_to_defect_now := false;
       END_IF;

   ELSE
       #go_to_defect_now := false;
   END_IF;


   #xdefect_inc_was := #xBdefect_inc;
   #xdefect_dec_was := #xBdefect_dec;
END_REGION

REGION Network 2 (SCL)
   IF #xDefect_Save AND NOT #xDefect_Save_was THEN
       IF #DEFECTS_DB.N < #DEFECTS_DB.N_max THEN
           #DEFECTS_DB.pos_AR[#DEFECTS_DB.N] := "_MAIN_DB".Mot_Positions;
           #DEFECTS_DB.N := #DEFECTS_DB.N + 1;
       ELSE
           #xyBeepDone := true;
       END_IF;
   END_IF;

   #xDefect_Save_was := #xDefect_Save;


   IF #xDefectsClearAll AND NOT #xDefectsClearAll_was THEN
       #DEFECTS_DB.N := 0;
       #DEFECTS_DB.i := 0;

   END_IF;
   #xDefectsClearAll_was := #xDefectsClearAll;
END_REGION
END_FUNCTION_BLOCK

FUNCTION_BLOCK "_ML2_ts_block1"   // FB49, FBD
{ S7_Optimized_Access := 'TRUE' }
VERSION : 0.1
// stored: AutoNumber true, IsIECCheckEnabled false, IsRetainMemResEnabled false, MemoryReserve 100, SetENOAutomatically false, UDAEnableTagReadback false
   VAR_INPUT
      R_ALL : Bool;
      SwAuto : Bool;
      AutoRuning : Bool;
      Arrived : Bool;
      R_SeimAuto : Bool;
      CLK_Spot : Bool;
      CLK_Defect : Bool;
      CLK_Home : Bool;
      CLK_Load : Bool;
      CLK_Control2 : Bool;
      CLK_Control1 : Bool;
   END_VAR
   VAR_OUTPUT
      Q0_Auto : Bool;
      q0_AutoWaiting : Bool;
      Q0_SemiAuto : Bool;
      P1_Spot : Bool;
      Q1_Spot : Bool;
      P2_Defect : Bool;
      Q2_Defect : Bool;
      P3_Home : Bool;
      Q3_Home : Bool;
      P4_Load : Bool;
      Q4_Load : Bool;
      P5_Control1 : Bool;
      Q5_Control1 : Bool;
      P6_Control2 : Bool;
      Q6_control2 : Bool;
      Q99_none : Bool;
      Q99_Any : Bool;
   END_VAR
   VAR
      memarrived : Bool;
      reset_Qs : Bool;
      last_button_stands_Instance { S7_SetPoint := 'True'} : "last_button_stands";
      Q_integer { S7_SetPoint := 'True'} : Int;
      trDefect { S7_SetPoint := 'True'} : R_TRIG;
      trSpot { S7_SetPoint := 'True'} : R_TRIG;
      bsu_Spot { S7_SetPoint := 'True'} : "_ML2_ts_block1_subunit";
      bsu_Defect { S7_SetPoint := 'True'} : "_ML2_ts_block1_subunit";
      bsuHome { S7_SetPoint := 'True'} : "_ML2_ts_block1_subunit";
      bsu_load { S7_SetPoint := 'True'} : "_ML2_ts_block1_subunit";
      bsuControl1 { S7_SetPoint := 'True'} : "_ML2_ts_block1_subunit";
      bsuControl2 { S7_SetPoint := 'True'} : "_ML2_ts_block1_subunit";
   END_VAR
   VAR CONSTANT
      Qi0_off : Int := 0;
      Qi1_Spot : Int := 1;
      Qi2_Defect : Int := 2;
      Qi3Home : Int := 3;
      Qi4Load : Int := 4;
      Qi5Control1 : Int := 5;
      Qi6Control2 : Int := 6;
   END_VAR
   VAR_TEMP   // added for the SCL form of the ladder/FBD networks
      _w1 : Bool;
   END_VAR
BEGIN

REGION Network 2
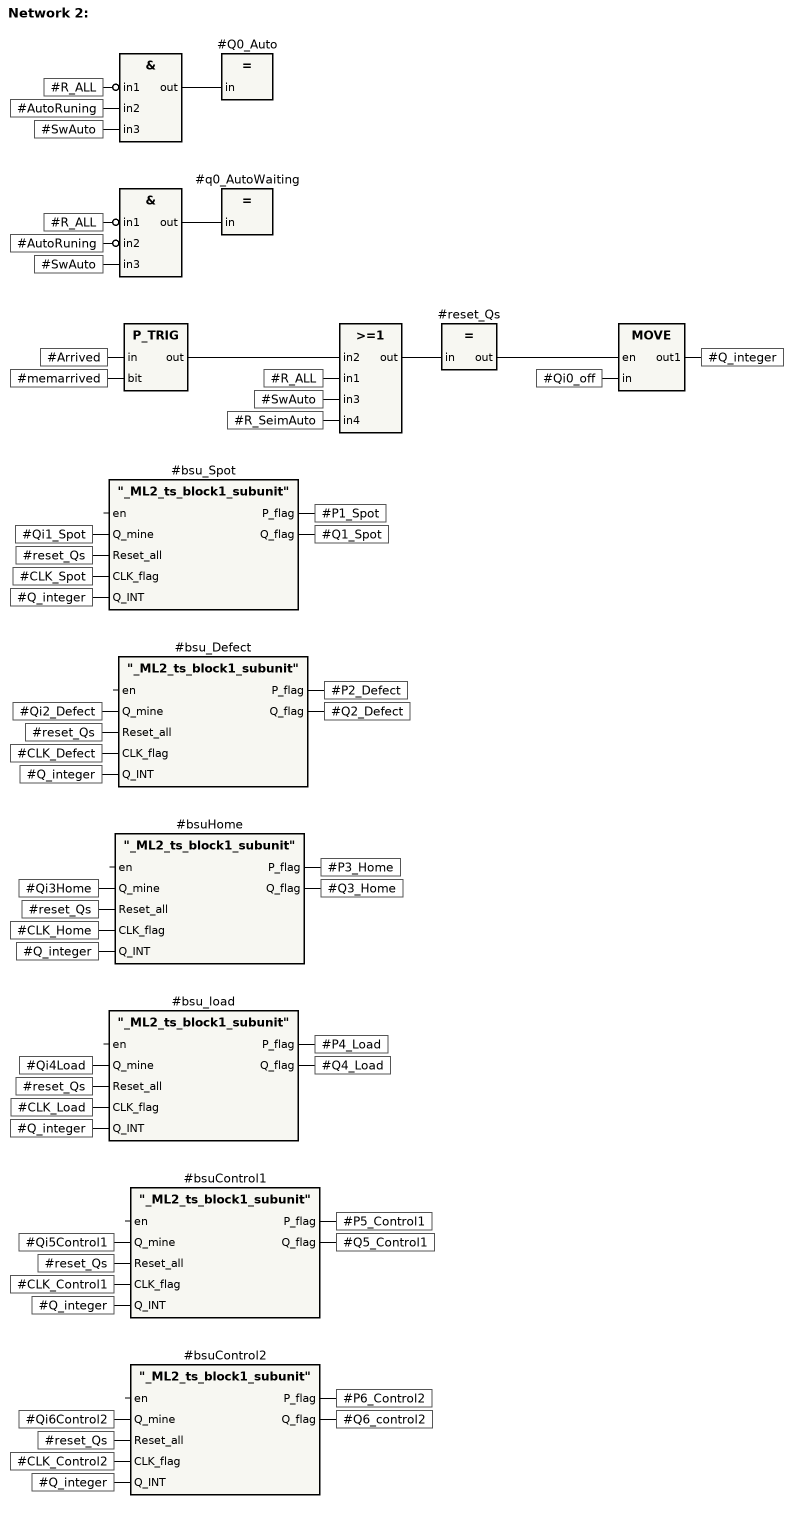
   #Q0_Auto := NOT #R_ALL AND #AutoRuning AND #SwAuto;
   #q0_AutoWaiting := NOT #R_ALL AND NOT #AutoRuning AND #SwAuto;
   #_w1 := #Arrived AND NOT #memarrived;   // rising edge
   #memarrived := #Arrived;
   #reset_Qs := #_w1 OR #R_ALL OR #SwAuto OR #R_SeimAuto;
   IF #reset_Qs THEN #Q_integer := #Qi0_off; END_IF;
   #bsu_Spot(Q_mine := #Qi1_Spot,   // "_ML2_ts_block1_subunit"
             Reset_all := #reset_Qs,
             CLK_flag := #CLK_Spot,
             Q_INT := #Q_integer,
             P_flag => #P1_Spot,
             Q_flag => #Q1_Spot);
   #bsu_Defect(Q_mine := #Qi2_Defect,   // "_ML2_ts_block1_subunit"
               Reset_all := #reset_Qs,
               CLK_flag := #CLK_Defect,
               Q_INT := #Q_integer,
               P_flag => #P2_Defect,
               Q_flag => #Q2_Defect);
   #bsuHome(Q_mine := #Qi3Home,   // "_ML2_ts_block1_subunit"
            Reset_all := #reset_Qs,
            CLK_flag := #CLK_Home,
            Q_INT := #Q_integer,
            P_flag => #P3_Home,
            Q_flag => #Q3_Home);
   #bsu_load(Q_mine := #Qi4Load,   // "_ML2_ts_block1_subunit"
             Reset_all := #reset_Qs,
             CLK_flag := #CLK_Load,
             Q_INT := #Q_integer,
             P_flag => #P4_Load,
             Q_flag => #Q4_Load);
   #bsuControl1(Q_mine := #Qi5Control1,   // "_ML2_ts_block1_subunit"
                Reset_all := #reset_Qs,
                CLK_flag := #CLK_Control1,
                Q_INT := #Q_integer,
                P_flag => #P5_Control1,
                Q_flag => #Q5_Control1);
   #bsuControl2(Q_mine := #Qi6Control2,   // "_ML2_ts_block1_subunit"
                Reset_all := #reset_Qs,
                CLK_flag := #CLK_Control2,
                Q_INT := #Q_integer,
                P_flag => #P6_Control2,
                Q_flag => #Q6_control2);
END_REGION

REGION Network 3
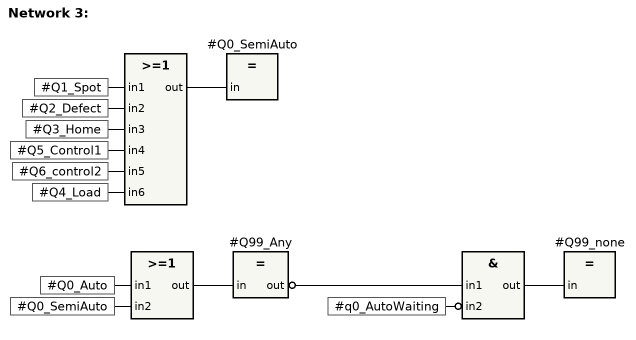
   #Q0_SemiAuto := #Q1_Spot OR #Q2_Defect OR #Q3_Home OR #Q5_Control1 OR #Q6_control2 OR #Q4_Load;
   #_w1 := #Q0_Auto OR #Q0_SemiAuto;
   #Q99_Any := #_w1;
   #Q99_none := NOT #_w1 AND NOT #q0_AutoWaiting;
END_REGION
END_FUNCTION_BLOCK

FUNCTION_BLOCK "_ML2_ts_block1_subunit"   // FB69, FBD
{ S7_Optimized_Access := 'TRUE' }
VERSION : 0.1
// stored: AutoNumber true, IsIECCheckEnabled false, IsRetainMemResEnabled false, MemoryReserve 100, SetENOAutomatically false, UDAEnableTagReadback false
   VAR_INPUT
      Q_mine : Int;
      Reset_all : Bool;
      CLK_flag : Bool;
   END_VAR
   VAR_OUTPUT
      P_flag : Bool;
      Q_flag : Bool;
   END_VAR
   VAR_IN_OUT
      Q_INT : Int;
   END_VAR
   VAR
      tr { S7_SetPoint := 'True'} : R_TRIG;
   END_VAR
BEGIN

REGION Network 1
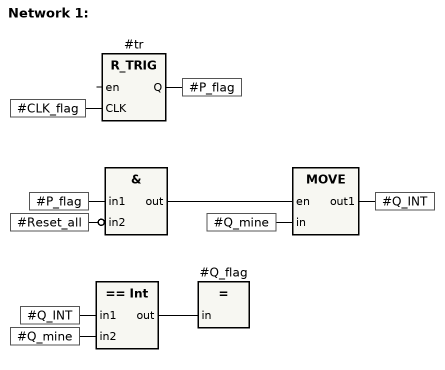
   #tr(CLK := #CLK_flag, Q => #P_flag);   // R_TRIG
   IF #P_flag AND NOT #Reset_all THEN #Q_INT := #Q_mine; END_IF;
   #Q_flag := #Q_INT = #Q_mine;
END_REGION
END_FUNCTION_BLOCK

FUNCTION_BLOCK "last_button_stands"
{ S7_Optimized_Access := 'TRUE' }
VERSION : 0.1
   VAR_INPUT 
      Reset_all : Bool;
      pt : Time := T#100ms;
   END_VAR

   VAR_OUTPUT 
      safe1 : Bool;
      safe2 : Bool;
      safe3 : Bool;
      safe4 : Bool;
      safe5 : Bool;
      safe6 : Bool;
      safe7 : Bool;
      safe8 : Bool;
      none_selected : Bool;
      change_trig { ExternalAccessible := 'False'; ExternalVisible := 'False'; ExternalWritable := 'False'} : Bool;
      reset_or_ch_or_none : Bool;
   END_VAR

   VAR_IN_OUT 
      B1 : Bool;
      B2 : Bool;
      B3 : Bool;
      B4 : Bool;
      B5 : Bool;
      B6 : Bool;
      B7 : Bool;
      B8 : Bool;
   END_VAR

   VAR 
      t {InstructionName := 'R_TRIG'; LibVersion := '1.0'} : Array[1..#N] of R_TRIG;
      B { S7_SetPoint := 'True'} : Array[1..#N] of Bool;
      S { S7_SetPoint := 'True'} : Array[1..#N] of Bool;
      tp { S7_SetPoint := 'False'} : "tp_peter";
   END_VAR

   VAR_TEMP 
      i : Int;
      j : Int;
   END_VAR

   VAR CONSTANT 
      N : Int := 8;
   END_VAR


BEGIN
	#B[1] := #B1;
	#B[2] := #B2;
	#B[3] := #B3;
	#B[4] := #B4;
	#B[5] := #B5;
	#B[6] := #B6;
	#B[7] := #B7;
	#B[8] := #B8;
	
	IF #Reset_all THEN
	    FOR #i := 1 TO #N DO
	        #B[#i] := false;
	    END_FOR;
	ELSE
	    FOR #i := 1 TO #N DO
	        #t[#i](CLK := #B[#i]);
	    END_FOR;
	    
	    
	    
	    FOR #i := 1 TO #N DO
	        IF #t[#i].Q THEN
	            FOR #j := 1 TO #N DO
	                IF #i <> #j THEN
	                    #B[#j] := false;
	                END_IF;
	            END_FOR;
	        END_IF;
	    END_FOR;
	    
	    #change_trig := false;
	    
	    FOR #i := 1 TO #N DO
	        #change_trig := #change_trig OR #t[#i].Q;
	    END_FOR;
	    #tp(CLK := #change_trig,
	        pt := #pt);
	    
	    
	    FOR #i := 1 TO #N DO
	        #S[#i] := #B[#i] AND NOT #tp.Q;
	    END_FOR;
	END_IF;
	
	IF #Reset_all THEN
	    #none_selected := false;
	ELSE
	    #none_selected := TRUE;
	    FOR #i := 1 TO #N DO
	        #none_selected := #none_selected AND NOT #B[#i];
	    END_FOR;
	    #none_selected := #none_selected;
	END_IF;
	
	#reset_or_ch_or_none := #none_selected OR  #change_trig OR #Reset_all;
	
	#B1 := #B[1];
	#B2 := #B[2];
	#B3 := #B[3];
	#B4 := #B[4];
	#B5 := #B[5];
	#B6 := #B[6];
	#B7 := #B[7];
	#B8 := #B[8];
	
	
	
	
	#safe1 := #S[1];
	#safe2 := #S[2];
	#safe3 := #S[3];
	#safe4 := #S[4];
	#safe5 := #S[5];
	#safe6 := #S[6];
	#safe7 := #S[7];
	#safe8 := #S[8];
	
END_FUNCTION_BLOCK

FUNCTION_BLOCK "tp_peter"   // FB40, LAD
{ S7_Optimized_Access := 'TRUE' }
VERSION : 0.1
// stored: AutoNumber true, IsIECCheckEnabled false, IsRetainMemResEnabled false, MemoryReserve 100, SetENOAutomatically false, UDAEnableTagReadback false
   VAR_INPUT
      CLK : Bool;
      pt : Time := T#100ms;
   END_VAR
   VAR_OUTPUT
      Q : Bool;
   END_VAR
   VAR
      was : Bool;
      ton { S7_SetPoint := 'True'} : TON_TIME;
   END_VAR
BEGIN

REGION Network 1
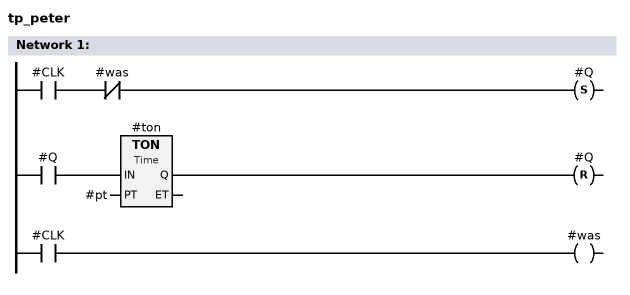
   RUNG wire#powerrail
      Contact( #CLK )
      I_Contact( #was )
      S_Coil( #Q )
   END_RUNG
   RUNG wire#powerrail
      Contact( #Q )
      { S7_Templates := "time_type := Time" } #ton.TON(pt := #pt, et =>)
      R_Coil( #Q )
   END_RUNG
   RUNG wire#powerrail
      Contact( #CLK )
      Coil( #was )
   END_RUNG
   // the same network as SCL:
   IF #CLK AND NOT #was THEN #Q := TRUE; END_IF;
   #ton(IN := #Q, PT := #pt);   // TON
   IF #ton.Q THEN #Q := FALSE; END_IF;
   #was := #CLK;
END_REGION
END_FUNCTION_BLOCK

FUNCTION_BLOCK "ER_WORD"
{ S7_Optimized_Access := 'TRUE' }
VERSION : 0.1
   VAR_INPUT 
      ignoreNewEr : Bool;
      ak { S7_HiddenAssignment := 'Show'} : Bool;
      x0 { S7_HiddenAssignment := 'HideIfNoParamAssigned'} : Bool;
      x1 { S7_HiddenAssignment := 'HideIfNoParamAssigned'} : Bool;
      x2 { S7_HiddenAssignment := 'HideIfNoParamAssigned'} : Bool;
      x3 { S7_HiddenAssignment := 'HideIfNoParamAssigned'} : Bool;
      x4 { S7_HiddenAssignment := 'HideIfNoParamAssigned'} : Bool;
      x5 { S7_HiddenAssignment := 'HideIfNoParamAssigned'} : Bool;
      x6 { S7_HiddenAssignment := 'HideIfNoParamAssigned'} : Bool;
      x7 { S7_HiddenAssignment := 'HideIfNoParamAssigned'} : Bool;
      x8 { S7_HiddenAssignment := 'HideIfNoParamAssigned'} : Bool := false;
      x9 { S7_HiddenAssignment := 'HideIfNoParamAssigned'} : Bool := false;
      x10 { S7_HiddenAssignment := 'HideIfNoParamAssigned'} : Bool := false;
      x11 { S7_HiddenAssignment := 'HideIfNoParamAssigned'} : Bool := false;
      x12 { S7_HiddenAssignment := 'HideIfNoParamAssigned'} : Bool := false;
      x13 { S7_HiddenAssignment := 'HideIfNoParamAssigned'} : Bool := false;
      x14 { S7_HiddenAssignment := 'HideIfNoParamAssigned'} : Bool := false;
      x15 { S7_HiddenAssignment := 'HideIfNoParamAssigned'} : Bool := false;
      selfreset0 { S7_HiddenAssignment := 'HideIfNoParamAssigned'} : Bool;
      selfreset1 { S7_HiddenAssignment := 'HideIfNoParamAssigned'} : Bool;
      selfreset2 { S7_HiddenAssignment := 'HideIfNoParamAssigned'} : Bool;
      selfreset3 { S7_HiddenAssignment := 'HideIfNoParamAssigned'} : Bool;
      selfreset4 { S7_HiddenAssignment := 'HideIfNoParamAssigned'} : Bool;
      selfreset5 { S7_HiddenAssignment := 'HideIfNoParamAssigned'} : Bool;
      selfreset6 { S7_HiddenAssignment := 'HideIfNoParamAssigned'} : Bool;
      selfreset7 { S7_HiddenAssignment := 'HideIfNoParamAssigned'} : Bool;
      selfreset8 { S7_HiddenAssignment := 'HideIfNoParamAssigned'} : Bool;
      selfreset9 { S7_HiddenAssignment := 'HideIfNoParamAssigned'} : Bool;
      selfreset10 { S7_HiddenAssignment := 'HideIfNoParamAssigned'} : Bool;
      selfreset11 { S7_HiddenAssignment := 'HideIfNoParamAssigned'} : Bool;
      selfreset12 { S7_HiddenAssignment := 'HideIfNoParamAssigned'} : Bool;
      selfreset13 { S7_HiddenAssignment := 'HideIfNoParamAssigned'} : Bool;
      selfreset14 { S7_HiddenAssignment := 'HideIfNoParamAssigned'} : Bool;
      selfreset15 { S7_HiddenAssignment := 'HideIfNoParamAssigned'} : Bool;
   END_VAR

   VAR_OUTPUT 
      _w : Word;
      er : Bool;
      count : Int;
      "a_er[0]" : Bool;
      "a_er[1]" : Bool;
      "a_er[2]" : Bool;
      "a_er[3]" : Bool;
      "a_er[4]" : Bool;
      "a_er[5]" : Bool;
      "a_er[6]" : Bool;
      "a_er[7]" : Bool;
      "a_er[8]" : Bool;
      "a_er[9]" : Bool;
      "a_er[10]" : Bool;
      "a_er[11]" : Bool;
      "a_er[12]" : Bool;
      "a_er[13]" : Bool;
      "a_er[14]" : Bool;
      "a_er[15]" : Bool;
   END_VAR

   VAR 
      a_er : Array[0..15] of Bool;
      a_x : Array[0..15] of Bool;
      a_is_self_reset : Array[0..15] of Bool;
   END_VAR

   VAR_TEMP 
      i : Int;
   END_VAR


BEGIN
	
	
	
	
	
	
	#a_x[0] := #x0;
	#a_x[1] := #x1;
	#a_x[2]:= #x2;
	#a_x[3]:= #x3;
	#a_x[4]:= #x4;
	#a_x[5]:= #x5;
	#a_x[6]:= #x6;
	#a_x[7]:= #x7;
	#a_x[8]:= #x8;
	#a_x[9]:= #x9;
	#a_x[10]:= #x10;
	#a_x[11]:= #x11;
	#a_x[12]:= #x12;
	#a_x[13]:= #x13;
	#a_x[14]:= #x14;
	#a_x[15]:= #x15;
	
	#a_is_self_reset[0] := #selfreset0;
	#a_is_self_reset[1] := #selfreset1;
	#a_is_self_reset[2] := #selfreset2;
	#a_is_self_reset[3] := #selfreset3;
	#a_is_self_reset[4] := #selfreset4;
	#a_is_self_reset[5] := #selfreset5;
	#a_is_self_reset[6] := #selfreset6;
	#a_is_self_reset[7] := #selfreset7;
	#a_is_self_reset[8] := #selfreset8;
	#a_is_self_reset[9] := #selfreset9;
	#a_is_self_reset[10] := #selfreset10;
	#a_is_self_reset[11] := #selfreset11;
	#a_is_self_reset[12] := #selfreset12;
	#a_is_self_reset[13] := #selfreset13;
	#a_is_self_reset[14] := #selfreset14;
	#a_is_self_reset[15] := #selfreset15;
	
	
	
	
	IF NOT #ignoreNewEr THEN
	    FOR #i := 0 TO 15 DO
	        IF #a_x[#i] THEN
	            #a_er[#i] := TRUE;
	        END_IF;
	    END_FOR;
	END_IF;
	
	
	
	#count := 0;
	FOR #i := 0 TO 15 DO
	    IF #a_er[#i] THEN
	        #count := #count + 1;
	    END_IF;
	END_FOR;
	
	#_w.%X0 := #a_er[00];
	#_w.%X1 := #a_er[01];
	#_w.%X2 := #a_er[02];
	#_w.%X3 := #a_er[03];
	#_w.%X4 := #a_er[04];
	#_w.%X5 := #a_er[05];
	#_w.%X6 := #a_er[06];
	#_w.%X7 := #a_er[07];
	#_w.%X8 := #a_er[08];
	#_w.%X9 := #a_er[09];
	#_w.%X10 := #a_er[10];
	#_w.%X11 := #a_er[11];
	#_w.%X12 := #a_er[12];
	#_w.%X13 := #a_er[13];
	#_w.%X14 := #a_er[14];
	#_w.%X15 := #a_er[15];
	#er := #_w > 0;
	
	
	FOR #i := 0 TO 15 DO
	    IF #ak THEN
	        #a_er[#i] := false;
	    END_IF;
	END_FOR;
	
	FOR #i := 0 TO 15 DO
	    IF #a_is_self_reset[#i] AND NOT #a_x[#i] THEN
	        #a_er[#i] := false;
	    END_IF;
	END_FOR;
	
	
	#"a_er[0]" := #a_er[00];
	#"a_er[1]" := #a_er[01];
	#"a_er[2]" := #a_er[02];
	#"a_er[3]" := #a_er[03];
	#"a_er[4]" := #a_er[04];
	#"a_er[5]" := #a_er[05];
	#"a_er[6]" := #a_er[06];
	#"a_er[7]" := #a_er[07];
	#"a_er[8]" := #a_er[08];
	#"a_er[9]" := #a_er[09];
	#"a_er[10]" := #a_er[10];
	#"a_er[11]" := #a_er[11];
	#"a_er[12]" := #a_er[12];
	#"a_er[13]" := #a_er[13];
	#"a_er[14]" := #a_er[14];
	#"a_er[15]" := #a_er[15];
	
END_FUNCTION_BLOCK

FUNCTION "ERRORS_WARNINGS_main" : Void   // FC32, FBD
{ S7_Optimized_Access := 'TRUE' }
VERSION : 0.1
// stored: AutoNumber true, IsIECCheckEnabled false, SetENOAutomatically false, UDAEnableTagReadback false
   VAR_TEMP
      er_count : Int;
      wn_count : Int;
      loc_count : Int;
      loc_c : Bool;
   END_VAR
BEGIN

REGION Network 1
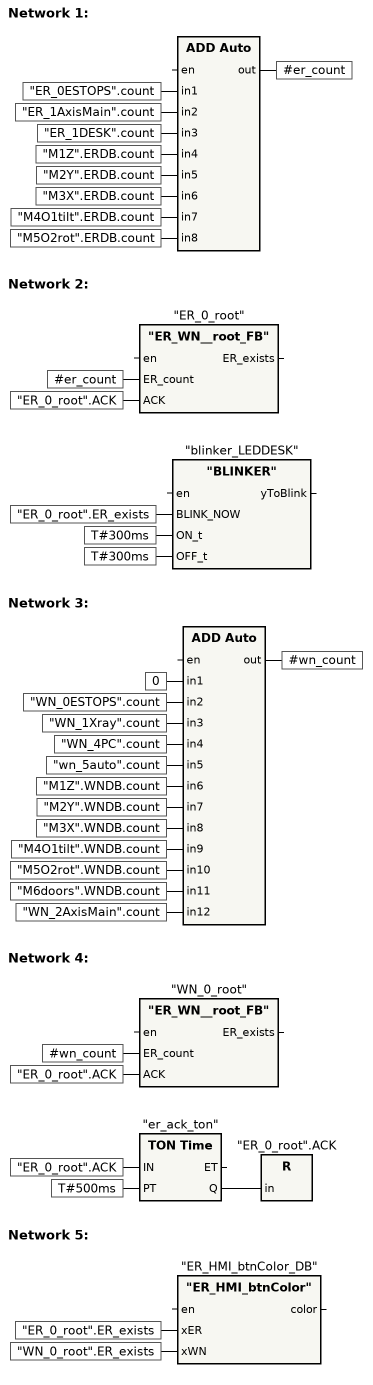
   #er_count := "ER_0ESTOPS".count + "ER_1AxisMain".count + "ER_1DESK".count + "M1Z".ERDB.count + "M2Y".ERDB.count + "M3X".ERDB.count + "M4O1tilt".ERDB.count + "M5O2rot".ERDB.count;
END_REGION

REGION Network 2
   "ER_0_root"(ER_count := #er_count, ACK := "ER_0_root".ACK);   // "ER_WN__root_FB"
   "blinker_LEDDESK"(BLINK_NOW := "ER_0_root".ER_exists, ON_t := T#300ms, OFF_t := T#300ms);   // "BLINKER"
END_REGION

REGION Network 3
   #wn_count := 0 + "WN_0ESTOPS".count + "WN_1Xray".count + "WN_4PC".count + "wn_5auto".count + "M1Z".WNDB.count + "M2Y".WNDB.count + "M3X".WNDB.count + "M4O1tilt".WNDB.count + "M5O2rot".WNDB.count + "M6doors".WNDB.count + "WN_2AxisMain".count;
END_REGION

REGION Network 4
   "WN_0_root"(ER_count := #wn_count, ACK := "ER_0_root".ACK);   // "ER_WN__root_FB"
   "er_ack_ton".TON(IN := "ER_0_root".ACK, PT := T#500ms);
   IF "er_ack_ton".Q THEN "ER_0_root".ACK := FALSE; END_IF;
END_REGION

REGION Network 5
   "ER_HMI_btnColor_DB"(xER := "ER_0_root".ER_exists, xWN := "WN_0_root".ER_exists);   // "ER_HMI_btnColor"
END_REGION

REGION Network 6
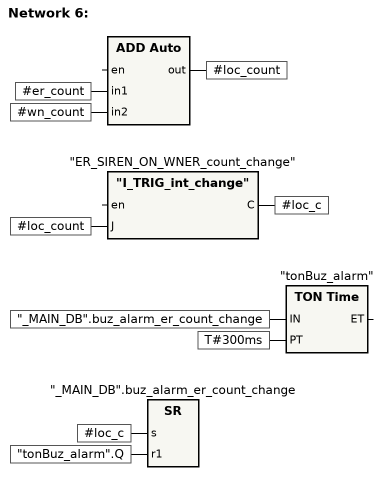
   #loc_count := #er_count + #wn_count;
   "ER_SIREN_ON_WNER_count_change"(J := #loc_count, C => #loc_c);   // "I_TRIG_int_change"
   "tonBuz_alarm".TON(IN := "_MAIN_DB".buz_alarm_er_count_change, PT := T#300ms);
   IF #loc_c THEN
       "_MAIN_DB".buz_alarm_er_count_change := TRUE;   // SR flip-flop
   END_IF;
   IF "tonBuz_alarm".Q THEN "_MAIN_DB".buz_alarm_er_count_change := FALSE; END_IF;
END_REGION
END_FUNCTION

FUNCTION_BLOCK "ER_WN__root_FB"   // FB64, LAD
{ S7_Optimized_Access := 'TRUE' }
VERSION : 0.1
// stored: AutoNumber true, IsIECCheckEnabled false, IsRetainMemResEnabled false, MemoryReserve 100, SetENOAutomatically false, UDAEnableTagReadback false
   VAR_INPUT
      ER_count : Int;
      ACK : Bool;
   END_VAR
   VAR_OUTPUT
      ER_exists : Bool;
   END_VAR
BEGIN

REGION Network 1
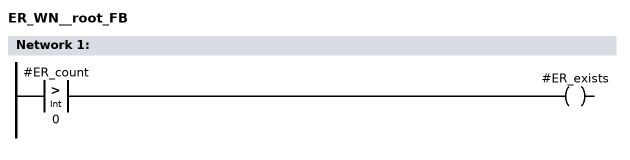
   RUNG wire#powerrail
      { S7_Templates := "SrcType := Int" } GT_Contact(in1 := #ER_count, in2 := 0)
      Coil( #ER_exists )
   END_RUNG
   // the same network as SCL:
   #ER_exists := #ER_count > 0;
END_REGION
END_FUNCTION_BLOCK

FUNCTION_BLOCK "BLINKER"   // FB30, LAD
{ S7_Optimized_Access := 'TRUE' }
VERSION : 0.1
// stored: AutoNumber true, IsIECCheckEnabled false, IsRetainMemResEnabled false, MemoryReserve 100, SetENOAutomatically false, UDAEnableTagReadback false
   VAR_INPUT
      BLINK_NOW : Bool;
      ON_t : Time := T#10s;
      OFF_t : Time := T#10s;
   END_VAR
   VAR_OUTPUT
      yToBlink : Bool;
   END_VAR
   VAR
      tON_DB { S7_SetPoint := 'True'} : TON_TIME;
      tOFF_DB { S7_SetPoint := 'True'} : TON_TIME;
      off_mem { S7_SetPoint := 'True'} : Bool;
   END_VAR
   VAR_TEMP   // added for the SCL form of the ladder/FBD networks
      _w1 : Bool;
   END_VAR
BEGIN

REGION Network 1
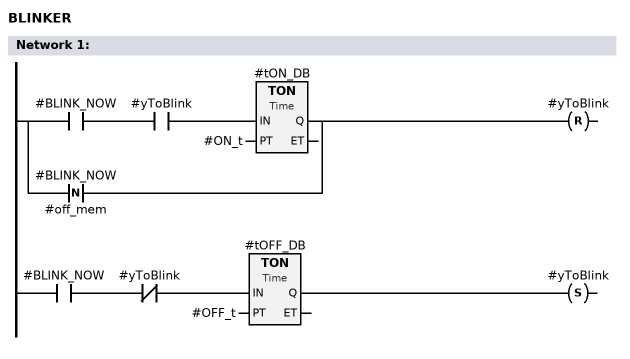
   RUNG wire#powerrail
      Contact( #BLINK_NOW )
      Contact( #yToBlink )
      { S7_Templates := "time_type := Time" } #tON_DB.TON(pt := #ON_t, et =>)
      wire#w1
      R_Coil( #yToBlink )
   END_RUNG
   RUNG wire#powerrail
      N_Contact(operand := #BLINK_NOW, bit := #off_mem)
   END_RUNG wire#w1
   RUNG wire#powerrail
      Contact( #BLINK_NOW )
      I_Contact( #yToBlink )
      { S7_Templates := "time_type := Time" } #tOFF_DB.TON(pt := #OFF_t, et =>)
      S_Coil( #yToBlink )
   END_RUNG
   // the same network as SCL:
   #tON_DB(IN := #BLINK_NOW AND #yToBlink, PT := #ON_t);   // TON
   #_w1 := NOT #BLINK_NOW AND #off_mem;   // falling edge of #BLINK_NOW
   #off_mem := #BLINK_NOW;
   IF #tON_DB.Q OR #_w1 THEN #yToBlink := FALSE; END_IF;
   #tOFF_DB(IN := #BLINK_NOW AND NOT #yToBlink, PT := #OFF_t);   // TON
   IF #tOFF_DB.Q THEN #yToBlink := TRUE; END_IF;
END_REGION
END_FUNCTION_BLOCK

FUNCTION_BLOCK "ER_HMI_btnColor"   // FB2, FBD
{ S7_Optimized_Access := 'TRUE' }
VERSION : 0.1
// stored: AutoNumber true, IsIECCheckEnabled false, IsRetainMemResEnabled false, MemoryReserve 100, SetENOAutomatically false, UDAEnableTagReadback false
   VAR_INPUT
      xER : Bool;
      xWN : Bool;
   END_VAR
   VAR_OUTPUT
      color : Int;
   END_VAR
   VAR CONSTANT
      c0clear : Int := 0;
      c1alarm : Int := 1;
      c2warning : Int := 2;
   END_VAR
BEGIN

REGION Network 1 (SCL)
   IF #xER THEN
       #color := #c1alarm;
   ELSIF #xWN THEN
       #color := #c2warning;
   ELSE
       #color := #c0clear;
   END_IF;
END_REGION
END_FUNCTION_BLOCK

FUNCTION_BLOCK "I_TRIG_int_change"   // FB52, FBD
{ S7_Optimized_Access := 'TRUE' }
VERSION : 0.1
// stored: AutoNumber true, IsIECCheckEnabled false, IsRetainMemResEnabled false, MemoryReserve 100, SetENOAutomatically false, UDAEnableTagReadback false
   VAR_INPUT
      J : Int;
   END_VAR
   VAR_OUTPUT
      C : Bool;
   END_VAR
   VAR
      J_was : Int;
   END_VAR
BEGIN

REGION Network 1
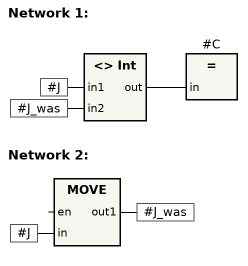
   #C := #J <> #J_was;
END_REGION

REGION Network 2
   #J_was := #J;
END_REGION
END_FUNCTION_BLOCK

FUNCTION "cab_main" : Void   // FC1, FBD
{ S7_Optimized_Access := 'TRUE' }
VERSION : 0.1
// stored: AutoNumber true, IsIECCheckEnabled false, SetENOAutomatically false, UDAEnableTagReadback false
   VAR_TEMP
      erCOM_A1 : Bool;
      wnDelay : Bool;
      er_нуевыеБлокировки : Bool;
      pt : Time;
   END_VAR
BEGIN

REGION Network 3
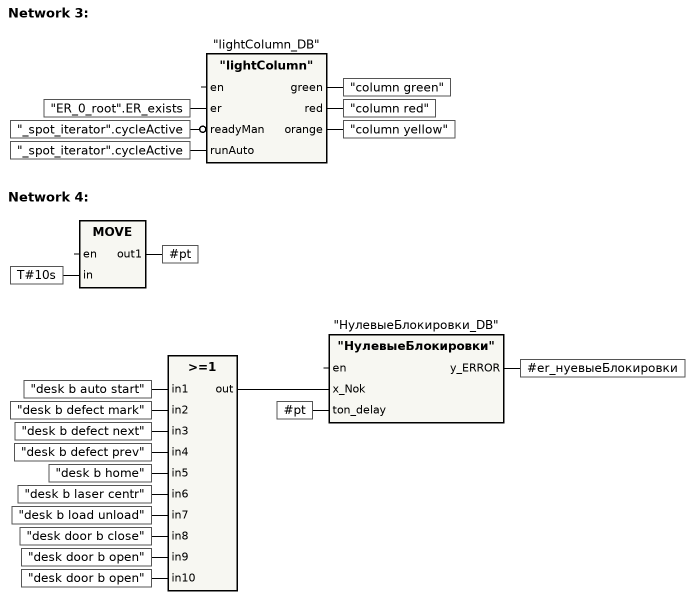
   "lightColumn_DB"(er := "ER_0_root".ER_exists,   // "lightColumn"
                    readyMan := NOT "_spot_iterator".cycleActive,
                    runAuto := "_spot_iterator".cycleActive,
                    green => "column green",
                    red => "column red",
                    orange => "column yellow");
END_REGION

REGION Network 4
   #pt := T#10s;
   "НулевыеБлокировки_DB"(x_Nok := "desk b auto start" OR "desk b defect mark" OR "desk b defect next" OR "desk b defect prev" OR "desk b home" OR "desk b laser centr" OR "desk b load unload" OR "desk door b close" OR "desk door b open" OR "desk door b open",   // "НулевыеБлокировки"
                          ton_delay := #pt,
                          y_ERROR => #er_нуевыеБлокировки);
END_REGION

REGION Network 5
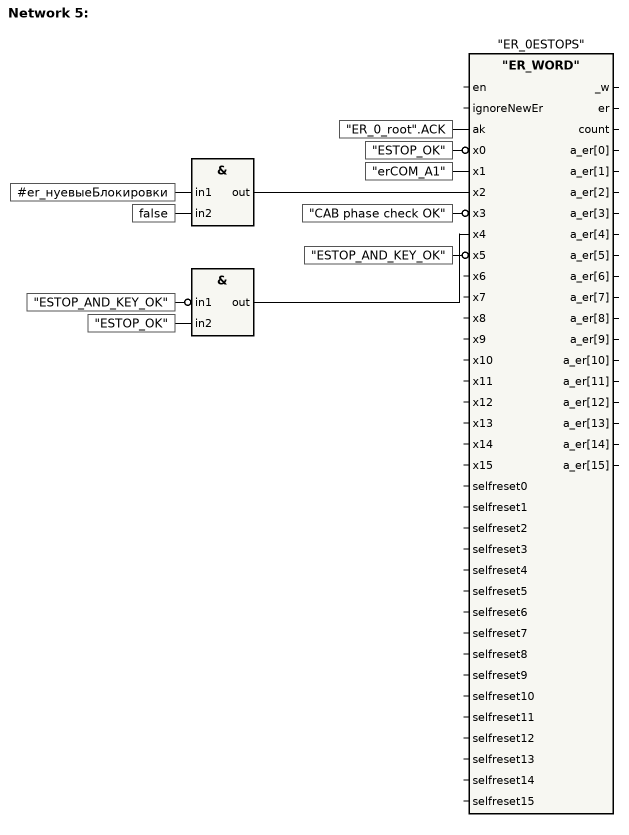
   "ER_0ESTOPS"(ak := "ER_0_root".ACK,   // "ER_WORD"
                x0 := NOT "ESTOP_OK",
                x1 := "erCOM_A1",
                x2 := #er_нуевыеБлокировки AND false,
                x3 := NOT "CAB phase check OK",
                x4 := NOT "ESTOP_AND_KEY_OK" AND "ESTOP_OK",
                x5 := NOT "ESTOP_AND_KEY_OK");
END_REGION

REGION Network 6
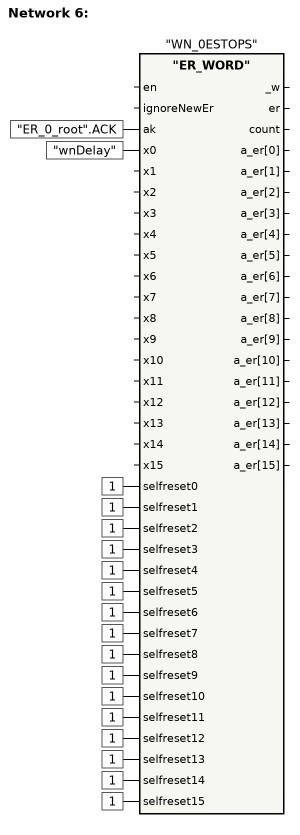
   "WN_0ESTOPS"(ak := "ER_0_root".ACK,   // "ER_WORD"
                x0 := "wnDelay",
                selfreset0 := 1,
                selfreset1 := 1,
                selfreset2 := 1,
                selfreset3 := 1,
                selfreset4 := 1,
                selfreset5 := 1,
                selfreset6 := 1,
                selfreset7 := 1,
                selfreset8 := 1,
                selfreset9 := 1,
                selfreset10 := 1,
                selfreset11 := 1,
                selfreset12 := 1,
                selfreset13 := 1,
                selfreset14 := 1,
                selfreset15 := 1);
END_REGION
END_FUNCTION

FUNCTION_BLOCK "lightColumn"   // FB44, FBD
{ S7_Optimized_Access := 'TRUE' }
VERSION : 0.1
// stored: AutoNumber true, IsIECCheckEnabled false, IsRetainMemResEnabled false, MemoryReserve 100, SetENOAutomatically false, UDAEnableTagReadback false
   VAR_INPUT
      er : Bool;
      readyMan : Bool;
      runAuto : Bool;
   END_VAR
   VAR_OUTPUT
      green : Bool;
      red : Bool;
      orange : Bool;
   END_VAR
BEGIN

REGION Network 1
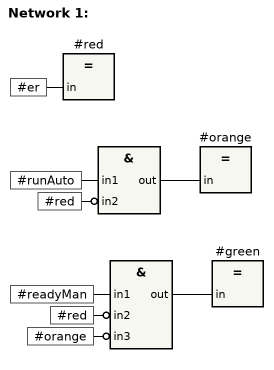
   #red := #er;
   #orange := #runAuto AND NOT #red;
   #green := #readyMan AND NOT #red AND NOT #orange;
END_REGION
END_FUNCTION_BLOCK

FUNCTION_BLOCK "НулевыеБлокировки"   // FB39, FBD
{ S7_Optimized_Access := 'TRUE' }
VERSION : 0.1
// stored: AutoNumber true, IsIECCheckEnabled false, IsRetainMemResEnabled false, MemoryReserve 100, SetENOAutomatically false, UDAEnableTagReadback false
   VAR_INPUT
      x_Nok : Bool;
   END_VAR
   VAR_OUTPUT
      y_ERROR : Bool := true;
   END_VAR
   VAR_IN_OUT
      ton_delay : Time := T#1s;
   END_VAR
   VAR
      IEC_Timer_0_Instance { S7_SetPoint := 'True'} : TON_TIME;
   END_VAR
   VAR_TEMP
      ton_elapsed : Bool;
   END_VAR
BEGIN

REGION Network 1
